    IF _eDeformStep > E_DeformationStep.nothing AND _bCamReady AND _bTeachOk THEN      // start only if previous started
      (*done during attach: 
      IF _eDeformStep < E_DeformationStep.cameraStarted THEN
        // start cam on ct
        LogLvl(Lvl:=E_LogSeverity.Debug, Msg:=F_Concat2('Start Camera with mode: ', TO_STRING(_iActiveCam.eCameraMode)));
        _pAttachedCt^.StartCamera(eCameraMode:=_iActiveCam.eCameraMode, fFeatureGrid:=_fFeatureGrid);
      *)
			IF _eDeformStep >= E_DeformationStep.cameraStarted AND _bCamStarted THEN
        // run update on ct
        // stream points
        streamPoints();
        // superview abort cases
      END_IF
      
      // NOTE: Release() is done in CamDone() method
    ELSE
      IF _bCamStarted THEN
        // error on camera while started
        LogError('Abort Camera while it was started');
			END_IF
      // release because cam not ready or pior worker not done its job
      Release(_pAttachedCt^);   // release head container
		END_IF

END_IF

// call messages
fbMsg_CamNotAvailable    (bI_Status:=bCamNotAvailable);
fbMsg_CamModeNotSupported(bI_Status:=bCamModeNotSupported);
fbMsg_CamNoConnection    (bI_Status:=NOT _bConnectionOk);
END_METHOD

END_FUNCTION_BLOCK

// ---- POUs/Print/DefGrid/FB_WorkerDefGrid.TcPOU
FUNCTION_BLOCK ABSTRACT FB_WorkerDefGrid EXTENDS FB_Worker
VAR_OUTPUT
  bError            : BOOL;                           // an error is active
  nError            : UDINT;                          // error code if error active, =0 else
END_VAR
VAR
  // config
  _pMsgConfigExt    : POINTER TO ST_MSG_CONFIG;       // external message config (puc message interface)
  _fPrintResolution : LREAL := 1;                     // print(head) resolution in [dpi]
  _fSubPxResolution : LREAL := 1;                     // SubPixel resolution [SubPx], resolution factor (fI_PrintResolution*fI_SubPxResolution=>Output resolution
  _name             : STRING;                         // Worker name
  _sVisuName        : STRING := 'VISU_WorkerDefGrid'; // Worker visu instance name
  _pEcSrc           : POINTER TO T_ErrSrc;            // Error source definition

  // job
  _bJobActive       : BOOL;                           // a job is active
  // ct
  _bAttached        : BOOL;                           // one ct is attached
  _pAttachedCt      : POINTER TO FB_ContainerDefGrid; // currently attached container (HEAD)
  _pNewAttached     : POINTER TO FB_ContainerDefGrid; // last attached container (as return value of Attach() (TAIL))
  _pNewAttachedHdlData : POINTER TO ST_WorkerDefGrid_CTData;  // pointer to handling data for last attached
  _bSupportParallelCT : BOOL := FALSE;                // support for parallel CTs (else avoid attach while one connected).
  _nAttachedCTs     : UDINT;                          // Number of currently attached CTs
  _nHeadCtId        : DINT;                           // ID of CT at Attached Head
  _pAttachedCTList  : ARRAY[nLowerIndexCTList..nUpperIndexCTList] OF POINTER TO FB_ContainerDefGrid;    // current attached CTs
  _stAttachedCTData : ARRAY[nLowerIndexCTList..nUpperIndexCTList] OF ST_WorkerDefGrid_CTData;           // additional "handling" data per attached CT
  // position control
  fCtPosition       : LREAL;     // Container position relative to worker position
  _bForceRelease    : BOOL;                           // Manually force a ct release

  // view
  nGridRowStart, nGridColStart: UDINT := 0;
END_VAR
VAR_STAT
  // static variables, SAME for ALL Workers
  _pCTM             : POINTER TO FB_CTManagerDefGrid;             // "Global" Container Manager
  _fCtSecurityReleasePos : LREAL := 0;                // [SubPx] position where to release current ct at last (security release)
END_VAR
VAR PERSISTENT
  _fWorkerPosition  : LREAL;                          // [m] worker distance to X0 (position from X0) (CT creation X0 and domain)
END_VAR
VAR CONSTANT
  // list size
  nLowerIndexCTList : UDINT := 1;
  nUpperIndexCTList : UDINT := 4; 
END_VAR

(*
  Generic abort implementation of DefGrid CT.
*)
METHOD Abort
VAR_INPUT
  iCT       : I_CT;
  sReason   : STRING;
END_VAR
VAR
  _pCt   : POINTER TO FB_ContainerDefGrid;
  eStep     : E_DeformationStep;
END_VAR
IF iCT = 0 AND _pAttachedCt <> 0 THEN             // no ct given and check if one is attached 
  _pCt := _pAttachedCt;
ELSIF getCtInst(iCT:=iCT, pCT=>_pCt) = 0 THEN     // get specific container from given interface
  RETURN; 
END_IF

IF _pCt = 0 THEN RETURN; END_IF
  
// abort CT
  // Do generic known aborts on CT
  // - Deformation
  _pCt^.getDeformationStatus(eDStep=>eStep);
  IF eStep >= E_DeformationStep.nothing THEN
    _pCt^.AbortDeformation(sReason:=sReason, Src:=_pEcSrc^, bHideLog:=FALSE);
  
END_IF
END_METHOD

METHOD PROTECTED  Attach : BOOL
VAR_INPUT
  iCT       : I_CT;            (*container at triggered event position*)
END_VAR
VAR
  i : UDINT;
END_VAR
Attach := FALSE;

IF iCT = 0 THEN
  LogError(Msg:='attach failed -> not ct given');
  
ELSIF bWorkerEnable THEN  // worker enabled
  
  IF getCtInst(iCT:=iCT, pCT=>_pNewAttached) <> 0 THEN    // get specific container
    // add to list ()
    IF push(pNewCT:=_pNewAttached) THEN 
      LogLvl(Lvl:=E_LogSeverity.Debug, Msg:=F_Concat4('Attach CT[', TO_STRING(_nAttachedCTs), ']: ', _pNewAttached^.print(0)));
      Attach:=TRUE;                                 // attach new
    END_IF
  ELSE
    LogError(Msg:='attach failed: could not get CT instance');
  END_IF

ELSIF NOT bWorkerEnable AND _nAttachedCTs > 0 THEN // disabled and already a CT attached
  // force release all attached CT, and ignore attach
  LogLvl(Lvl:=E_LogSeverity.Debug, Msg:='Worker disabled flush list of all attached CT');
  WHILE _nAttachedCTs > 0 DO
    Release(iCT:=_pAttachedCt^);
	END_WHILE

ELSIF NOT bWorkerEnable AND _pAttachedCt = 0 THEN  
  ;   // nothing to do, ignore attach

ELSE      // unspecified (error)case just log it
  LogError(Msg:='not tracked case');
END_IF


// ok to attach
END_METHOD

{attribute 'monitoring':='call'}
PROPERTY bAttached : BOOL
GET
bAttached := _bAttached;
END_GET
END_PROPERTY

{attribute 'monitoring':='call'}
PROPERTY fPosition : LREAL
GET
fPosition := _fWorkerPosition;
END_GET
SET
_fWorkerPosition := fPosition;  // [m] save position
END_SET
END_PROPERTY

(*
  Get specific container from interface.
  Returns specific container in return value and output parameter.
*)
METHOD INTERNAL getCtInst : POINTER TO FB_ContainerDefGrid
VAR_INPUT
  iCT              : I_CT;                         (*container at triggered event position*)
END_VAR
VAR_OUTPUT
  pCT              : POINTER TO FB_ContainerDefGrid;
END_VAR
IF NOT bInitialized THEN RETURN; END_IF
IF _pCTM = 0 THEN RETURN; END_IF

pCT := 0;
getCtInst := _pCTM^.GetContainerInstance(iCT);   // get real ct fb inst
IF getCtInst <> 0 THEN
  pCT := getCtInst;   // OK all good
ELSE
  LogError(Msg:='specific container not found');
END_IF
END_METHOD

(*
  Get relative position to this worker (relative to track position)
*)
METHOD getPosRelToAttach : DINT
VAR_INPUT
  iCT : I_CT;
END_VAR
// relative position to X0 - tracking offset of this worker
getPosRelToAttach := iCT.GetPosRel(iTracker:=_iCTTracker) - _nTrackOffset;
END_METHOD

METHOD Init
VAR_INPUT
  pMsgConfig : POINTER TO ST_MSG_CONFIG;         // message config
  fPrintResolution : LREAL := 1;                 // print(head) resolution in [dpi]
  fSubPxResolution : LREAL := 1;                 // SubPixel resolution [SubPx], resolution factor (fI_PrintResolution*fI_SubPxResolution=>Output resolution)
  bParallelCT : BOOL;                            // Support parallel processing of CTs
END_VAR
VAR

END_VAR
_bAttached := 0;
_pAttachedCt := 0;
_nAttachedCTs := 0;

IF _pCTM = 0 THEN LogError(Msg:='Init: invalid parameter'); RETURN; END_IF

// save config
_pMsgConfigExt := pMsgConfig;
_fPrintResolution := fPrintResolution;
_fSubPxResolution := fSubPxResolution;
_fCtSecurityReleasePos := 0;
_bSupportParallelCT := bParallelCT;

setName('');

// init error source reference
_pEcSrc := ErrorCodes.fbErrCodeMngr.registerErrSource(
  nLocId := 0,
  aInstPath := InstanceName,
  aLocDescr := _name
);
IF _pEcSrc = 0 THEN LogError('could not register error source'); END_IF

bInitialized := TRUE;
END_METHOD

METHOD ABSTRACT mJobStart
VAR_INPUT
	sJobDef	: CalmarCompPrint.I_JobDefinition;
END_VAR
// implement in parent class
END_METHOD

METHOD ABSTRACT mJobStop
VAR_INPUT
	sStatus	: CalmarCompPrint.I_JobStatus;
END_VAR
END_METHOD

PROPERTY pCTM : POINTER TO FB_CTManagerDefGrid
GET
pCTM := _pCTM;
END_GET
SET
_pCTM := pCTM;
END_SET
END_PROPERTY

METHOD PRIVATE pull : BOOL
VAR_INPUT
  pRemCT : POINTER TO FB_ContainerDefGrid;
END_VAR
VAR_OUTPUT
  nRemIndex : DINT := 0;
END_VAR
VAR
  i                : DINT;
  Index            : DINT;
  LowerIndex       : DINT := 1;
END_VAR
IF _nAttachedCTs = 0 THEN LogError('Release: but no CT is attached'); RETURN; END_IF

// -- find if ct is in attached list
Index := -1;
FOR i:= TO_DINT(nLowerIndexCTList) TO TO_DINT(nLowerIndexCTList + _nAttachedCTs - 1) DO
  IF _pAttachedCTList[i] = pRemCT THEN
    Index := i;
    EXIT;     // found
  END_IF
END_FOR
IF Index = -1 THEN LogError('Release: ct inst not found in list'); RETURN; END_IF

// do stop CT callback if removing first
IF Index = TO_DINT(nLowerIndexCTList) THEN StopCT(pCtDefGrid:=pRemCT); END_IF

// compress list
IF Index >= TO_DINT(nLowerIndexCTList) AND Index < TO_DINT(nUpperIndexCTList) THEN
  // - ct references
  MEMMOVE(              // shift all above entries down
    destAddr := ADR( _pAttachedCTList[Index] ), 
    srcAddr  := ADR( _pAttachedCTList[Index + 1] ), 
    n        := DINT_TO_UDINT(SIZEOF(_pAttachedCTList[LowerIndex]) * (UDINT_TO_DINT(_nAttachedCTs) - Index - 1 + LowerIndex))
  );
  _pAttachedCTList[nUpperIndexCTList] := 0;     // erase last(compressed) list entry
  // - ct handling data
  MEMMOVE(              // shift all above entries down
    destAddr := ADR( _stAttachedCTData[Index] ), 
    srcAddr  := ADR( _stAttachedCTData[Index + 1] ), 
    n        := DINT_TO_UDINT(SIZEOF(_stAttachedCTData[LowerIndex]) * (UDINT_TO_DINT(_nAttachedCTs) - Index - 1 + LowerIndex))
  );
  MEMSET(destAddr:=ADR(_stAttachedCTData[nUpperIndexCTList]), fillByte:=0, n:=SIZEOF(_stAttachedCTData[1]));  // erase last(compressed) list entry
END_IF
_pAttachedCTList[_nAttachedCTs] := 0;   // erase last element
MEMSET(destAddr:=ADR(_stAttachedCTData[_nAttachedCTs]), fillByte:=0, n:=SIZEOF(_stAttachedCTData[1]));  // erase last element
  
// remove
_nAttachedCTs := _nAttachedCTs - 1;   // remove one element

IF _nAttachedCTs > 0 THEN 
  // Start new HEAD
  _pAttachedCt := _pAttachedCTList[1];
  _bAttached := TRUE;
  StartCT(pCtDefGrid:=_pAttachedCt);
ELSE
  // CT list empty (no ct attached)
  _pAttachedCt := 0;
  _bAttached := 0;
END_IF

nRemIndex := Index;
pull := TRUE;
END_METHOD

METHOD PRIVATE push : BOOL
VAR_INPUT
  pNewCT : POINTER TO FB_ContainerDefGrid;
END_VAR
// checks
// - valid param
IF pNewCT = 0 THEN LogError('push: invalid pointer'); RETURN; END_IF
// - list full
IF _nAttachedCTs >= nUpperIndexCTList THEN  // list overflow no free element for processing
  LogError('Worker processing list full, ignore new CT');
  Abort(iCT:=pNewCT^, sReason:='attach failed - too many attached');  // abort new CT (no release because not yet attached)
  RETURN;
END_IF
// - only one CT allowed
IF _nAttachedCTs > 0 AND NOT _bSupportParallelCT THEN
  LogError(Msg:='another container already attached -> ignore new (set error)');
  Abort(iCT:=pNewCt^, sReason:='attach failed - no parallel support');  // abort new CT
END_IF

// add to list
_nAttachedCTs := _nAttachedCTs + 1;
_pAttachedCTList[_nAttachedCTs] := pNewCT;
MEMSET(destAddr:=ADR(_stAttachedCTData[_nAttachedCTs]), fillByte:=0, n:=SIZEOF(_stAttachedCTData[1]));  // clear additional data
_pNewAttachedHdlData := ADR(_stAttachedCTData[_nAttachedCTs]);   // select handling data for new attached ct 

// apply head
IF _nAttachedCTs = 1 THEN
  // set HEAD
  _pAttachedCt := _pAttachedCTList[nLowerIndexCTList];  
  _bAttached := TRUE;

  // start callback on HEAD
  StartCT(pCtDefGrid:=_pAttachedCt);
END_IF

push := TRUE;
END_METHOD

(*
  Release CT from Worker.
  :return: TRUE if CT was released, FALSE if no CT was registered 
*)
METHOD Release : BOOL
VAR_INPUT
  iCT              : I_CT;                         (*container at triggered event position*)
END_VAR
VAR
  nIdx             : DINT;
  pCT              : POINTER TO FB_ContainerDefGrid;
END_VAR
// remove CT -----------------------------------------------------
// -- get real instance
pCT := getCtInst(iCT:=iCT);
IF pCT = 0 THEN LogError('Release: could not find ct instance'); RETURN; END_IF

// remove and release CT
IF pull(pRemCT:=pCT, nRemIndex=>nIdx) THEN
  LogLvl(Lvl:=E_LogSeverity.Debug, Msg:=F_Concat4('Release CT[', TO_STRING(nIdx), '] ', pCt^.print(0)));
  Release := TRUE;  
END_IF
END_METHOD

(*
  Container will be released from tracker (destroyed) and not available anymore. 
*)
METHOD remove
VAR_INPUT
	(*container at triggered event position*)
	iCT	: I_CT;
END_VAR
SUPER^();

// nothing done
// We keep in internal WorkerList until work is done. CT will be removed from tracker.
END_METHOD

METHOD PRIVATE setName : BOOL
VAR_INPUT
  sName : STRING;
END_VAR
VAR
  nIdx : INT;
  bDone : BOOL;
END_VAR
IF sName = '' THEN
  // generate worker name
  _name := THIS^.InstanceName;
  WHILE NOT bDone DO
    nIdx := FIND(_name, '.');
    IF nIdx = 0 THEN bDone := TRUE; EXIT; 
    ELSE
      _name := RIGHT(_name,LEN(_name)-nIdx);
    END_IF 
  END_WHILE
ELSE
  _name := sName;  
END_IF
END_METHOD

METHOD PROTECTED StartCT
VAR_INPUT
 pCtDefGrid   : POINTER TO FB_ContainerDefGrid;
END_VAR
(* Override specific implementation in child class *)
END_METHOD

METHOD PROTECTED StopCT
VAR_INPUT
 pCtDefGrid   : POINTER TO FB_ContainerDefGrid;
END_VAR
(* Override specific implementation in child class *)
END_METHOD

METHOD  work
VAR
  i : UDINT;
  pCt : POINTER TO FB_ContainerDefGrid;
END_VAR
// set tracking offset
_nTrackOffset := F_MeterToSubPixel(fPosMeter:=fPosition, fResoSubPx:=_fPrintResolution*_fSubPxResolution);  // [pos domain] save position

//Work only with attached container
IF _nAttachedCTs = 0 THEN RETURN; END_IF

IF _pAttachedCt <> 0 AND_THEN _pAttachedCt^.pCT <> 0 THEN _nHeadCtId := _pAttachedCt^.pCT^.iId;
ELSE                                                      _nHeadCtId := 0; END_IF

FOR i:=nLowerIndexCTList TO nLowerIndexCTList + _nAttachedCTs - 1 DO
  pCt := _pAttachedCTList[i];

  // update CT position
  _stAttachedCTData[i].fPosRelToAttach := getPosRelToAttach(iCT:=pCt^);
  
  // release CT (manually)
  IF _bForceRelease THEN
    _bForceRelease := FALSE;
    pCt^.AbortDeformation(sReason:='Manually realease CT', Src:=_pEcSrc^, bHideLog:=FALSE);
    Release(iCT:=pCt^);

  // security release 
  ELSIF _fCtSecurityReleasePos > 0 AND (ABS(_stAttachedCTData[i].fPosRelToAttach) > _fCtSecurityReleasePos) THEN
    pCt^.AbortDeformation(sReason:=F_Concat2('Security released CT Id=', TO_STRING(pCt^.pCT^.iId)), Src:=_pEcSrc^, bHideLog:=FALSE);
    Release(iCT:=pCt^);
  END_IF

END_FOR
END_METHOD

END_FUNCTION_BLOCK

// ---- POUs/Print/DefGrid/FB_WorkerDefGrid_Deformation.TcPOU
FUNCTION_BLOCK FB_WorkerDefGrid_Deformation EXTENDS FB_WorkerDefGrid
VAR_INPUT
END_VAR
VAR_OUTPUT
END_VAR
VAR
  // references
  _iParamMediator : I_ParamMediator;
  
  //Worker specific configuration
  _nPrintUnitWidth            : UDINT;  // default print unit width [px]  
  _nImageWidthPx              : UDINT;  // size of the image (width)
  _nImageDepthPx              : UDINT;  // size of the image (depth)
  
  // -
  _bNewJob                    : BOOL;   // new job started 

  //Deformation status (per attached CT)
  _nDeformationProcPoints     : ARRAY[nLowerIndexCTList..nUpperIndexCTList] OF UDINT;  // available grid points on ct
  _nDeformationProcCols       : ARRAY[nLowerIndexCTList..nUpperIndexCTList] OF UDINT;  // number of already generated grid columns
  _eDeformStep                : ARRAY[nLowerIndexCTList..nUpperIndexCTList] OF E_DeformationStep;   // status deformation of ct
  _bDeformationError          : ARRAY[nLowerIndexCTList..nUpperIndexCTList] OF BOOL;   // status deformation of ct
  _bDeformationBusy           : ARRAY[nLowerIndexCTList..nUpperIndexCTList] OF BOOL;   // status deformation of ct
  _bDeformationDone           : ARRAY[nLowerIndexCTList..nUpperIndexCTList] OF BOOL;   // status deformation of ct
  _nDeformationErrorId        : ARRAY[nLowerIndexCTList..nUpperIndexCTList] OF UDINT;  // status deformation of ct
  _tDeformationExecutionTime  : ARRAY[nLowerIndexCTList..nUpperIndexCTList] OF TIME;   // status deformation of ct
  _bAborted                   : ARRAY[nLowerIndexCTList..nUpperIndexCTList] OF BOOL;   // status deformation of ct

  // ui
  eDeformTypeUi : E_DeformationType;
END_VAR 

VAR PERSISTENT
  _sDeformationGridSettings  : ST_DefGridSettings := (   // grid definition settings
                                  nGridPitchX:=GVL_Deformation.nC_DefaultGridPitch_X,   // this must match the hw config (in fpga)
                                  nGridPitchY:=GVL_Deformation.nC_DefaultGridPitch_Y,   // this must match the hw config (in fpag)
                                  eDeformationType:=E_DeformationType.NoDeformation
                             );
  _fDistToCam                : LREAL := 0.02;   // distance to cam worker 
END_VAR

METHOD PROTECTED  Attach : BOOL
VAR_INPUT
  iCT              : I_CT;                         (*container at triggered event position*)
END_VAR
VAR
  i : UDINT;
  bDeformErr : BOOL;
  eDeformStep : E_DeformationStep;
END_VAR
(*Please do enable externally in PrintModule
IF getCtInst(iCT:=iCT, pCT=>pCt) = 0 THEN    // get specific container
  RETURN;
END_IF

//-- (auto-) enable / disable worker based on mode (do before parent Attach(), is checked inside)
bWorkerEnable := _sDeformationGridSettings.eDeformationType <> E_DeformationType.NoDeformation 
                     AND SEL(pCt^.eCamMode > E_CameraMode.NoCorrection, FALSE, TRUE);
*)

// -- Attach
IF NOT SUPER^.Attach(iCT:=iCT) THEN
  RETURN;
END_IF

// Additional worker checks
IF _pNewAttached = 0 THEN RETURN; END_IF

// - Additional worker checks
bDeformErr := _pNewAttached^.getDeformationStatus(eDStep=>eDeformStep);   // get latest status 
  
// - deformation started? and no deformation error so far
IF bDeformErr OR eDeformStep < E_DeformationStep.cameraStarted THEN
  Release(iCT:=iCT);  // nothing to do anymore

  // - job is valid?
ELSIF _pNewAttached^.pJob = 0 OR NOT _bJobActive THEN
  _pNewAttached^.AbortDeformation(sReason:='No valid job', Src:=_pEcSrc^, bHideLog:=FALSE);
  Release(iCT:=iCT);
  
// - did camera start?  
(*ELSIF eDeformStep < E_DeformationStep.cameraStarted THEN
  _pNewAttached^.AbortDeformation(sReason:='Prio steps did not start', Src:=_pEcSrc^);
  Release(iCT:=iCT);
*)
  
// - OK attach
ELSE
  // checks
  IF eDeformStep < E_DeformationStep.cameraStarted THEN LogWarning('Sub-optimal timing, camera did not yet start'); END_IF
  // start deformation
  _pNewAttached^.StartDeformation(
    sDefGridSettings:=_sDeformationGridSettings, 
    fStartDeformationPos:=getPosRelToAttach(iCT)/_fSubPxResolution   // [px]
  );
  Attach := TRUE;
END_IF
END_METHOD

METHOD InitWorkerDeformation : BOOL
VAR_INPUT
  nPrintUnitWidth : UDINT;
  iDefGridParamMediator : I_ParamMediator;
END_VAR
VAR
  i : UDINT;
END_VAR
IF NOT bInitialized THEN LogError('Base Worker not initialized! call init() before'); RETURN; END_IF
IF iDefGridParamMediator = 0 THEN bInitialized := FALSE; LogError('Invalid parameter, no valid param mediator'); RETURN; END_IF


// worker specific init
_nPrintUnitWidth := nPrintUnitWidth;
_iParamMediator := iDefGridParamMediator;
_bNewJob := FALSE;

FOR i:=nLowerIndexCTList TO nUpperIndexCTList DO
  _nDeformationProcPoints[i]     := 0;
  _nDeformationProcCols[i]       := 0;
  _eDeformStep[i]                := 0;
  _bDeformationError[i]          := 0;
  _bDeformationBusy[i]           := 0;
  _bDeformationDone[i]           := 0;
  _nDeformationErrorId[i]        := 0;
  _tDeformationExecutionTime[i]  := T#0S;
  _bAborted[i]                   := 0;
END_FOR
END_METHOD

METHOD mJobStart
VAR_INPUT
	sJobDef	: CalmarCompPrint.I_JobDefinition;
END_VAR
VAR
  sCamSettings : ST_CameraGridSettings;
END_VAR
// check and init invalid settings
IF _iParamMediator = 0 THEN LogError('no parameter mediator'); RETURN; END_IF
IF _sDeformationGridSettings.nGridPitchX = 0 THEN _sDeformationGridSettings.nGridPitchX:=GVL_Deformation.nC_DefaultGridPitch_X; LogError(F_Concat2('nGridPitchX not configured, set default=', TO_STRING(GVL_Deformation.nC_DefaultGridPitch_X))); END_IF
IF _sDeformationGridSettings.nGridPitchY = 0 THEN _sDeformationGridSettings.nGridPitchY:=GVL_Deformation.nC_DefaultGridPitch_Y; LogError(F_Concat2('nGridPitchY not configured, set default=', TO_STRING(GVL_Deformation.nC_DefaultGridPitch_Y))); END_IF
IF _nPrintUnitWidth = 0 THEN LogError('_nPrintUnitWidth not configured'); END_IF
IF fPosition = 0 THEN LogError('No valid Worker position: set it to WorkerCamera.fCameraToPrintOffset + 0.05; '); END_IF

// configuration
// calculate deformation  settings
// - save image y-offset (centered)
// - save image size
_nImageWidthPx := DINT_TO_UDINT(F_MeterToSubPixel(fPosMeter:=sJobDef.fImageWidth/1000, fResoSubPx:=_fPrintResolution));
_nImageDepthPx := DINT_TO_UDINT(F_MeterToSubPixel(fPosMeter:=sJobDef.fImageDepth/1000, fResoSubPx:=_fPrintResolution));
_sDeformationGridSettings.nGridImageOffsetY := LIMIT(0, ((_nPrintUnitWidth - _nImageWidthPx)) / 2, (_nPrintUnitWidth));  // TODO: if you can get this value from PUC use the other one to have a consistent image shift value 

// - calc grid size and number of points
(*
  Use image width / depth in px divide by GridPitch in X/Y to do a ceil(always next bigger integer).
  +1 -> Because Grid starts at 0 until the calculated numbers we have one point more [0, 1, 2, 3] = 4 points (not 3) 
*)
IF _sDeformationGridSettings.nGridPitchX > 0 AND _sDeformationGridSettings.nGridPitchY > 0 THEN
  _sDeformationGridSettings.nGridSizeX := F_Ceil(val:=UDINT_TO_LREAL(_nImageDepthPx)/_sDeformationGridSettings.nGridPitchX) + 1;
  _sDeformationGridSettings.nGridSizeY := F_Ceil(val:=UDINT_TO_LREAL(_nImageWidthPx + _sDeformationGridSettings.nGridImageOffsetY)/_sDeformationGridSettings.nGridPitchY) + 1;
END_IF
_sDeformationGridSettings.nGridPoints :=  _sDeformationGridSettings.nGridSizeX * _sDeformationGridSettings.nGridSizeY;

sCamSettings := _iParamMediator.sCameraGridSettings;
_sDeformationGridSettings.eDeformationType := sCamSettings.eDeformationType;   // apply deformation mode (for ui)
eDeformTypeUi := _sDeformationGridSettings.eDeformationType;

_bJobActive := TRUE;
END_METHOD

METHOD  mJobStop
VAR_INPUT
	sStatus	: CalmarCompPrint.I_JobStatus;
END_VAR
_bJobActive := FALSE;
END_METHOD

(*
  Release CT from Worker.
  :return: TRUE if CT was released, FALSE if no CT was registered 
*)
METHOD Release : BOOL
VAR_INPUT
  iCT              : I_CT;                         (*container at triggered event position*)
END_VAR
VAR
  i                : DINT;
  Index            : DINT;
  LowerIndex       : DINT := 1;
  pCt              : POINTER TO FB_ContainerDefGrid;
  eStep            : E_DeformationStep;
END_VAR
IF iCT = 0 OR _nAttachedCTs = 0 THEN RETURN; END_IF

// release from deformation module
IF getCtInst(iCT:=iCT, pCT=>pCt) = 0 THEN LogError('Release: could not find ct instance'); RETURN; END_IF
IF _iParamMediator <> 0 THEN
  pCt^.getDeformationStatus(eDStep => estep);
  IF estep >= E_DeformationStep.createdScriptContainer THEN
    pCt^.StopScript(iCT:=iCT);
    //_pParamMediator^.ReleaseDeformationCT(iCT:=iCT);
  END_IF
END_IF

Release := SUPER^.Release(iCT:=iCT);
END_METHOD

PROPERTY sDeformationGridSettings : ST_DefGridSettings
GET
sDeformationGridSettings := _sDeformationGridSettings;
END_GET
END_PROPERTY

METHOD setupPosition
VAR
  sCamSettings : ST_CameraGridSettings;
END_VAR
IF _pAttachedCt <> 0 THEN RETURN; END_IF    // Update only without attached container

sCamSettings := _iParamMediator.sCameraGridSettings;

// set tracking offset
fPosition := sCamSettings.fDetectToCam + _fDistToCam;
END_METHOD

METHOD  work
VAR
  i : UDINT;
  pCT : POINTER TO FB_ContainerDefGrid;
END_VAR
//-----------------------------------------------------------
SUPER^.work();      // Parent implementation

setupPosition();    // Worker position update

// Work only with attached container (additional work to Base class)
FOR i:=nLowerIndexCTList TO nLowerIndexCTList + _nAttachedCTs - 1 DO
  pCt := _pAttachedCTList[i];
 
  // update deformation handler
  pCT^.UpdateDeformation(fPos:=_stAttachedCTData[i].fPosRelToAttach/_fSubPxResolution);  // pos in [px]
  
  // get status
  _bDeformationError[i] := pCt^.getDeformationStatus(eDStep => _eDeformStep[i], 
                            bBusy => _bDeformationBusy[i],
                            bDone => _bDeformationDone[i],
                            nErrorId => _nDeformationErrorId[i], 
                            tExecutionTime => _tDeformationExecutionTime[i],
                            bAborted => _bAborted[i]);
  _nDeformationProcPoints[i] := pCt^.nAvailableGridPoints;
  _nDeformationProcCols[i]   := pCt^.nAvailableGridCols;
     
  // Release container when all points have been processed or error
  IF _bDeformationDone[i] OR _bDeformationError[i] THEN
    // tag CT with error if deformation had an error
    IF _bDeformationError[i] THEN 
      IF NOT _bAborted[i] THEN
        pCt^.AbortDeformation(sReason:=F_Concat2('WorkerDeformation: ', EC_DefGrid.ecDefGrid_DefGridError.Desc), Src:=_pEcSrc^, bHideLog:=FALSE);
      //not needed ELSE
      //  pCt^.setError(ErrDef:=EC_DefGrid.ecDefGrid_DefGridError, Src:=_pEcSrc^);
      END_IF
    END_IF
    LogLvl(Lvl:=E_LogSeverity.Detail, Msg:=F_Concat4('Done with: CamP=',  TO_STRING(pCT^.nRegisteredCameraPoints), ' GridP=', TO_STRING(pCt^.nAvailableGridPoints)));
    Release(pCt^);
  END_IF
  
END_FOR
END_METHOD

END_FUNCTION_BLOCK

// ---- POUs/Print/DefGrid/FB_DropSpeedComp.TcPOU
FUNCTION_BLOCK FB_DropSpeedComp
VAR_INPUT
  fMasterSpeed         : LREAL; //[m/s]
  fDropTravelDistance  : LREAL; //[m]
END_VAR
VAR_OUTPUT
  fDropPlacementError  : LREAL;
END_VAR
VAR PERSISTENT
  _bEnable             : BOOL := TRUE;
  _fDropSpeed          : LREAL := 6;         //[m/s] DropSpeed compensation, drop speed
  _fDropSpeedDeadTime  : LREAL := 0.388889;  //[ms]  DropSpeed compensation, additional dead time
END_VAR
VAR
  bCalcDeadTime        : BOOL;
  fTestSpeed           : ARRAY[1..2] OF LREAL;  // [m/min] speed at which test was done [SpeedTest1, SpeedTest2]
  fTestDisplacement    : ARRAY[1..2] OF LREAL;  // [um] measured displacement after test [MesureTest1, MeasureTest2]
  fDiffSpeed : LREAL;
  fDiffPlace : LREAL;
END_VAR

(*Speed compensation*)
IF _bEnable AND (_fDropSpeed > 0) THEN
	fDropPlacementError :=  (  (fDropTravelDistance / _fDropSpeed)
                        + (_fDropSpeedDeadTime / 1000))             (*[s]*)
                        * fMasterSpeed;
ELSE
  fDropPlacementError := 0;
END_IF;

// calculate add/dead time
IF bCalcDeadTime THEN bCalcDeadTime := FALSE;
  calcDeadTime();
END_IF

{attribute 'monitoring':='call'}
PROPERTY bEnable : BOOL
GET
bEnable := _bEnable;
END_GET
SET
_bEnable := bEnable;
END_SET
END_PROPERTY

METHOD PRIVATE calcDeadTime : BOOL
VAR_INPUT
END_VAR
fDiffSpeed :=  ( fTestSpeed[2] - fTestSpeed[1] ) * 1/60;
fDiffPlace :=  ( fTestDisplacement[2] - fTestDisplacement[1] ) * 1/1_000_000;

IF fDiffSpeed <> 0 THEN   // avoid crash
  // calc time
  _fDropSpeedDeadTime := 
  (
      fDiffPlace      // displacement diff
    * 1/fDiffSpeed    // speed diff
  ) * 1000;           // [s] -> [ms]
ELSE
  F_LogError('DropSpeedComp invalid TestSpeed given -> DeadTime not updated');
END_IF


// reset entries
fTestSpeed[2] := fTestSpeed[1] := 0;
fTestDisplacement[2] := fTestDisplacement[1] := 0;
END_METHOD

{attribute 'monitoring':='call'}
PROPERTY fDropSpeed : LREAL
GET
fDropSpeed := _fDropSpeed;
END_GET
SET
_fDropSpeed := fDropSpeed;
END_SET
END_PROPERTY

{attribute 'monitoring':='call'}
PROPERTY fDropSpeedDeadTime : LREAL
GET
fDropSpeedDeadTime := _fDropSpeedDeadTime;
END_GET
SET
_fDropSpeedDeadTime := fDropSpeedDeadTime;
END_SET
END_PROPERTY

END_FUNCTION_BLOCK

// ---- POUs/Print/DefGrid/FB_FineAlignement.TcPOU
(*
  This fb handles mechanical print unit corrections.
  - a 4p grid distortion
  - print unit bar banana correction
  NOTE: temperature extention of whole printbar is still handled in camera
*)
FUNCTION_BLOCK FB_FineAlignement EXTENDS FB_BasePrint IMPLEMENTS I_GridPointCorrection
VAR
  // config
  _fPxResolution     : LREAL; // pixel resolution

  // corrections
  //-- 4 point PU deformation correction/distortion
  //    VISU setup point providing reference and correction (NOTE: persists settings internally)
  _fbPlcCorrPoints : ARRAY[1..4] OF FB_PointCorr;
  //-- banana correction
  _fT1 : LREAL;   // temperature 1
  _fT2 : LREAL;   // temperature 2
  _dx_middle : LREAL;  // correction in middle (for view only)
  _y_max : LREAL; // print unit width [mm]
  //-- PUC 4p correction
  _pAdsCam           : POINTER TO FB_ADS_CAMERA;  // camera interface PUC
  aPucPointNames : ARRAY[1..4] OF STRING := ['1','2','3','4'];
  
  // helper
  lCtr     : UDINT;
  
  // unit test & debug
  _bUT_4p, _bUT_banana, _bUT_4pPuc : BOOL;
  _sUTPoints_dx : ARRAY[0..nC_UT_cols, 0..nC_UT_rows] OF LREAL;
  _sUTPoints_dy : ARRAY[0..nC_UT_cols, 0..nC_UT_rows] OF LREAL;
  // 4pPUC
  bSelect : ARRAY[1..4] OF BOOL;
  bSelected : ARRAY[1..4] OF BOOL;
  nSelectedPoint : UDINT;
  bXPlus, bXMinus, bYPlus, bYMinus : BOOL;
END_VAR
VAR PERSISTENT
  //-- 4point correction
  _bEnable_4p    : BOOL := FALSE;
  _bEnablePuc_4p : BOOL := FALSE;
  //  persistence of points see: FB_PointCorr
  //-- banana correction
  _bEnable_banana : BOOL := FALSE;
  _e_max_per_deltaT : LREAL := 0.01;  // [mm/°C]  TODO: use from config
END_VAR
VAR CONSTANT
  // Unit test configuration
  nC_UT_cols : DINT := 6;   // for test only
  nC_UT_rows : DINT := 5;   // for test only
END_VAR

// cyclic caluclation and view updates
//        NOTE: deformation is happening in updateCorrection() callback

//-- 4p correction
//   visu overrides (limitation rectancular point definition)
_fbPlcCorrPoints[3].fX_Ref := _fbPlcCorrPoints[1].fX_Ref;
_fbPlcCorrPoints[4].fX_Ref := _fbPlcCorrPoints[2].fX_Ref;
_fbPlcCorrPoints[2].fY_Ref := _fbPlcCorrPoints[1].fY_Ref;
_fbPlcCorrPoints[4].fY_Ref := _fbPlcCorrPoints[3].fY_Ref;
//   update CorrectionPoints view elements
FOR lCtr := 1 TO 4 DO
  _fbPlcCorrPoints[lCtr](); 
END_FOR

//-- banana correction
// just calculate the dx in the middle of the PU, just for the VISU
calc_banana_correction(x_pos:=0, y_pos:=_y_max/(2*1000), fT1:=_fT1, fT2:=_fT2, dx_corr=>_dx_middle);
_dx_middle := _dx_middle * 1000; // [m] --> [mm] for visu

// Unit test
IF _bUT_4p THEN _bUT_4p := FALSE; _test_4p(); END_IF
IF _bUT_banana THEN _bUT_banana := FALSE; _test_banana(); END_IF
IF _bUT_4pPuc THEN _test_Puc4p(); END_IF

METHOD PRIVATE _test_4p
VAR
  sPoint : ST_DeformationPoint;
  nCol, nRow, nCrPoint : DINT;
  dx, dy : LREAL;       // correction in [m]
  dx_px, dy_px : DINT;  // correction in [px]
  pPUC_CorrPointsInd : POINTER TO ARRAY[1..4] OF ST_CORRECTION_POINT;
  
  nCorrectionX : ARRAY[1..4] OF REAL := [-0.25, -0.2, 0.35, 0.35];
  nCorrectionY : ARRAY[1..4] OF REAL := [-0.45, -0.3, -0.8, -0.65];
  nCorrectionPointX_PLC : ARRAY[1..4] OF REAL := [0, 1000,   0, 1000];
  nCorrectionPointY_PLC : ARRAY[1..4] OF REAL := [0,   0, 702, 702];
  nCorrectionPointX_PUC : ARRAY[1..4] OF REAL := [0, 671.99,   0, 671.99];
  nCorrectionPointY_PUC : ARRAY[1..4] OF REAL := [-0.0001666666, -0.0001666666, 754.2108, 754.2108];
END_VAR
// setup test correcton points location for PLC & PUC 4p testing
pPUC_CorrPointsInd := _pAdsCam^.pCorrectionPointsIndication;
IF pPUC_CorrPointsInd = 0 THEN F_Report_Error(ErrType:=EN_REPORT_ERROR_TYPE.Report_Error_0Pointer);  RETURN; END_IF

FOR nCrPoint:=1 TO 4 DO
  // correction point location
  // -- PLC
  _fbPlcCorrPoints[nCrPoint].fX_Ref := nCorrectionPointX_PLC[nCrPoint];
  _fbPlcCorrPoints[nCrPoint].fY_Ref := nCorrectionPointY_PLC[nCrPoint];
  // -- PUC  
  pPUC_CorrPointsInd^[nCrPoint].posx := nCorrectionPointX_PUC[nCrPoint];
  pPUC_CorrPointsInd^[nCrPoint].posy := nCorrectionPointY_PUC[nCrPoint];
  
  // point correction  
  // -- PLC
  _fbPlcCorrPoints[nCrPoint].fX := nCorrectionX[nCrPoint];
  _fbPlcCorrPoints[nCrPoint].fY := nCorrectionY[nCrPoint];
  // -- PUC
  pPUC_CorrPointsInd^[nCrPoint].x := nCorrectionX[nCrPoint];
  pPUC_CorrPointsInd^[nCrPoint].y := nCorrectionY[nCrPoint];
END_FOR

// generate internal test grid
FOR nCol:=0 TO nC_UT_cols DO
  FOR nRow:=0 TO nC_UT_rows DO
    sPoint.col := nCol;
    sPoint.row := nRow;
    sPoint.x_ref := nCol * TO_DINT(GVL_Deformation.nC_DefaultGridPitch_X);
    sPoint.y_ref := nRow * TO_DINT(GVL_Deformation.nC_DefaultGridPitch_Y);
    sPoint.dx := 0;   // no previous deformation
    sPoint.dy := 0;   // no previous deformation
    
    // calc 4p PLC correction and apply to point
    calc_4p_correction(
        x_pos:=F_SubPixelToMeter(lPosSubPx:=sPoint.x_ref, fResSubPx:=_fPxResolution), 
        y_pos:=F_SubPixelToMeter(lPosSubPx:=sPoint.y_ref, fResSubPx:=_fPxResolution), 
        dx_corr=>dx, 
        dy_corr=>dy);
    LogInfo(
      F_Concat4(
        '4p PLC: point:', 
        F_Concat4(' x=', TO_STRING(sPoint.x_ref), '/y=', TO_STRING(sPoint.y_ref)),
        F_Concat2(' dx=', TO_STRING(dx)),
        F_Concat2(' dy=', TO_STRING(dy))
      )
    );

    // --- store in table for verification with Excel caluculation
    dx_px := F_MeterToSubPixel(fPosMeter:=dx, fResoSubPx:=_fPxResolution);
    dy_px := F_MeterToSubPixel(fPosMeter:=dy, fResoSubPx:=_fPxResolution);
    // save corrected point
    _sUTPoints_dx[nCol, nRow] := dx_px;
    _sUTPoints_dy[nCol, nRow] := dy_px;
    // print corrected point
    LogInfo(
      F_Concat4(
        F_Concat4('[c/r] ', TO_STRING(sPoint.col), '/', TO_STRING(sPoint.row)),
        F_Concat7(' dx: ', TO_STRING(sPoint.dx), '>', TO_STRING(dx_px), ' (', TO_STRING(dx), ')'),
        F_Concat7(' dy: ', TO_STRING(sPoint.dy), '>', TO_STRING(dy_px), ' (', TO_STRING(dy), ')'),
        SEL(sPoint.dx<>dx_px OR sPoint.dy<>dy_px,'',' !!!')
      )
    );
    // ---------------------------------
    
    // calc 4p PUC correction and apply to point
    calc_PUC_4p_correction(
        x_pos:=F_SubPixelToMeter(lPosSubPx:=sPoint.x_ref, fResSubPx:=_fPxResolution), 
        y_pos:=F_SubPixelToMeter(lPosSubPx:=sPoint.y_ref, fResSubPx:=_fPxResolution), 
        dx_corr=>dx, 
        dy_corr=>dy);
    LogInfo(
      F_Concat4(
        '4p PUC: point:', 
        F_Concat4(' x=', TO_STRING(sPoint.x_ref), '/y=', TO_STRING(sPoint.y_ref)),
        F_Concat2(' dx=', TO_STRING(dx)),
        F_Concat2(' dy=', TO_STRING(dy))
      )
    );

  END_FOR  
END_FOR
END_METHOD

METHOD PRIVATE _test_banana
VAR
  sPoint : ST_DeformationPoint;
  nCol, nRow : DINT;
  dx, dy : LREAL;       // correction in [m]
  dx_px, dy_px : LREAL;  // correction in [px]
END_VAR
// generate internal grid
FOR nCol:=0 TO nC_UT_cols DO
  FOR nRow:=0 TO nC_UT_rows DO
    sPoint.col := nCol;
    sPoint.row := nRow;
    sPoint.x_ref := nCol * TO_DINT(GVL_Deformation.nC_DefaultGridPitch_X);
    sPoint.y_ref := nRow * TO_DINT(GVL_Deformation.nC_DefaultGridPitch_Y);
    sPoint.dx := 0;   // no previous deformation
    sPoint.dy := 0;   // no previous deformation
    
    // calc correction and apply to point
    calc_banana_correction(
        x_pos:=F_SubPixelToMeter(lPosSubPx:=sPoint.x_ref, fResSubPx:=_fPxResolution), 
        Y_pos:=F_SubPixelToMeter(lPosSubPx:=sPoint.y_ref, fResSubPx:=_fPxResolution),
        fT1 := 68,
        fT2 := 48, 
        dx_corr=>dx
    );
    dx_px := dx;
    dy_px := dy;
    // save corrected point (dx @y-pos)
    _sUTPoints_dx[nCol, nRow] := dx_px;
    _sUTPoints_dy[nCol, nRow] := F_SubPixelToMeter(lPosSubPx:=sPoint.y_ref, fResSubPx:=_fPxResolution)*1000;
    
    // print corrected point
    LogInfo(
      F_Concat4(
        F_Concat4('[c/r] ', TO_STRING(sPoint.col), '/', TO_STRING(sPoint.row)),
        F_Concat6(' dx: ', TO_STRING(sPoint.dx), '>', TO_STRING(TO_DINT(dx_px)), ' [', TO_STRING(dx)),
        F_Concat6('  dy: ', TO_STRING(sPoint.dy), '>', TO_STRING(TO_DINT(dy_px)), ' [', TO_STRING(dy)),
        SEL(sPoint.dx<>dx_px OR sPoint.dy<>dy_px,'',' !!!')
      )
    );
  END_FOR  
END_FOR
END_METHOD

METHOD PRIVATE _test_Puc4p
VAR
  i : UDINT;

  pPUC_CorrPointsInd : POINTER TO ARRAY[1..4] OF ST_CORRECTION_POINT;
  pPoint : POINTER TO ST_CORRECTION_POINT;
END_VAR
pPUC_CorrPointsInd := _pAdsCam^.pCorrectionPointsIndication;      // get points array from ADS
IF pPUC_CorrPointsInd = 0 THEN F_Report_Error(ErrType:=EN_REPORT_ERROR_TYPE.Report_Error_0Pointer);  RETURN; END_IF

// do selection
IF    bSelect[1] THEN bSelect[1]:=FALSE; MEMSET(destAddr:=ADR(bSelected), fillByte:=0, n:=SIZEOF(bSelected)); bSelected[1] := TRUE; nSelectedPoint:=1;
ELSIF bSelect[2] THEN bSelect[2]:=FALSE; MEMSET(destAddr:=ADR(bSelected), fillByte:=0, n:=SIZEOF(bSelected)); bSelected[2] := TRUE; nSelectedPoint:=2;
ELSIF bSelect[3] THEN bSelect[3]:=FALSE; MEMSET(destAddr:=ADR(bSelected), fillByte:=0, n:=SIZEOF(bSelected)); bSelected[3] := TRUE; nSelectedPoint:=3;
ELSIF bSelect[4] THEN bSelect[4]:=FALSE; MEMSET(destAddr:=ADR(bSelected), fillByte:=0, n:=SIZEOF(bSelected)); bSelected[4] := TRUE; nSelectedPoint:=4;
END_IF

IF    bSelected[1] THEN pPoint := ADR(pPUC_CorrPointsInd^[1]);
ELSIF bSelected[2] THEN pPoint := ADR(pPUC_CorrPointsInd^[2]);
ELSIF bSelected[3] THEN pPoint := ADR(pPUC_CorrPointsInd^[3]);
ELSIF bSelected[4] THEN pPoint := ADR(pPUC_CorrPointsInd^[4]);
ELSE                    pPoint := ADR(pPUC_CorrPointsInd^[1]);
END_IF

IF bXPlus  THEN bXPlus  := FALSE; pPoint^.x := pPoint^.x + 0.05; END_IF
IF bXMinus THEN bXMinus := FALSE; pPoint^.x := pPoint^.x - 0.05; END_IF
IF bYPlus  THEN bYPlus  := FALSE; pPoint^.y := pPoint^.y + 0.05; END_IF
IF bYMinus THEN bYMinus := FALSE; pPoint^.y := pPoint^.y - 0.05; END_IF
END_METHOD

(*
  Calculate grid point displacement for a distortion with 4 rectangular defined points.
  Uses 2-bilinear interpolation between the 4 rectancular reference points.
*)
METHOD PRIVATE calc_4p_correction : BOOL
VAR_INPUT
  x_pos   : LREAL;    // point x position [m]
  y_pos   : LREAL;    // point y position [m]
END_VAR
VAR_OUTPUT
  dx_corr : LREAL;    // point correction x [m]
  dy_corr : LREAL;    // point correction y [m]
END_VAR
VAR
  dx, dy : LREAL;     // difference between Calibration Points (rectangle)
  x1, x2, y1, y2 : LREAL;
  cx1, cx2, cy1, cy2 : LREAL;
  GPx, GPy : LREAL;
  CVx, CVy : LREAL;
  lErrCtr : UDINT;
END_VAR

// Grid point position
GPx := x_pos; 
GPy := y_pos;

// Interpolation in x
x1 := _fbPlcCorrPoints[1].fX_Ref / 1000;    // [mm -> m]
x2 := _fbPlcCorrPoints[2].fX_Ref / 1000;    // [mm -> m]
dx := x2-x1;
IF dx = 0 THEN (*F_Report_Error(ErrType:=EN_REPORT_ERROR_TYPE.Report_Error_0Pointer);*) RETURN; END_IF

cx1 := (x2-GPx)/dx * (_fbPlcCorrPoints[1].fX / 1000) + (GPx-x1)/dx * (_fbPlcCorrPoints[2].fX / 1000);
cx2 := (x2-GPx)/dx * (_fbPlcCorrPoints[3].fX / 1000) + (GPx-x1)/dx * (_fbPlcCorrPoints[4].fX / 1000);
cy1 := (x2-GPx)/dx * (_fbPlcCorrPoints[1].fY / 1000) + (GPx-x1)/dx * (_fbPlcCorrPoints[2].fY / 1000);
cy2 := (x2-GPx)/dx * (_fbPlcCorrPoints[3].fY / 1000) + (GPx-x1)/dx * (_fbPlcCorrPoints[4].fY / 1000);

// Interpolation in y
y1 := _fbPlcCorrPoints[1].fY_Ref / 1000;    // [mm -> m]
y2 := _fbPlcCorrPoints[3].fY_Ref / 1000;    // [mm -> m]
dy := y2-y1;
IF dy = 0 THEN (*F_Report_Error(ErrType:=EN_REPORT_ERROR_TYPE.Report_Error_0Pointer);*) RETURN; END_IF

// Calc interpolated 
CVx := (y2 - GPy)/dy * cx1 + (GPy-y1)/dy * cx2;
CVy := (y2 - GPy)/dy * cy1 + (GPy-y1)/dy * cy2;

// return accurate new correction only
dx_corr := CVx;
dy_corr := CVy;

calc_4p_correction := TRUE;
END_METHOD

(*
  Calculate grid point displacement for print unit banana deformation.
  2nd order approximation.
*)
METHOD PRIVATE calc_banana_correction : BOOL
VAR_INPUT
  x_pos   : LREAL;    // point x position [m]
  y_pos   : LREAL;    // point y position [m]
  fT1     : LREAL;    // temperature 1 [°C]
  fT2     : LREAL;    // temperature 2 [°C]
END_VAR
VAR_OUTPUT
  dx_corr : LREAL;    // point correction x [m]
END_VAR
VAR
  delta_T : LREAL;   // delta temperature
  e_max   : LREAL;   //
  a : LREAL;
  x_dash, y_dash : LREAL;
END_VAR
IF _y_max = 0 THEN RETURN; END_IF

x_dash := y_pos * 1000; // [m] -> [mm]

delta_T := fT2-fT1;
e_max   := delta_T * _e_max_per_deltaT;

a := 4 * e_max /  EXPT(_y_max, 2);
y_dash := a * EXPT(x_dash - (_y_max / 2), 2) - e_max;

// correction value
dx_corr := (y_dash / 1000);  // [mm] -> [m]

calc_banana_correction := TRUE;
END_METHOD

(*
  Calculate grid point displacement for a distortion with 4 rectangular defined points.
  Uses 2-bilinear interpolation between the 4 rectancular reference points.
*)
METHOD PRIVATE calc_PUC_4p_correction : BOOL
VAR_INPUT
  x_pos   : LREAL;    // point x position [m]
  y_pos   : LREAL;    // point y position [m]
END_VAR
VAR_OUTPUT
  dx_corr : LREAL;    // point correction x [m]
  dy_corr : LREAL;    // point correction y [m]
END_VAR
VAR
  dx, dy : LREAL;     // difference between Calibration Points (rectangle)
  x1, x2, y1, y2 : LREAL;
  cx1, cx2, cy1, cy2 : LREAL;
  GPx, GPy : LREAL;
  CVx, CVy : LREAL;
  lErrCtr : UDINT;
  
  pPUC_CorrPointsInd : POINTER TO ARRAY[1..4] OF ST_CORRECTION_POINT;
END_VAR
VAR CONSTANT
  fTranslateX : REAL := 1;
  fTranslateY : REAL := -1;
END_VAR
pPUC_CorrPointsInd := _pAdsCam^.pCorrectionPointsIndication;      // get points array from ADS
IF pPUC_CorrPointsInd = 0 THEN F_Report_Error(ErrType:=EN_REPORT_ERROR_TYPE.Report_Error_0Pointer);  RETURN; END_IF

// NOTE: the anchor points (poyx,posy) of the PUC points are set in WorkerCamera.mJobStart!

// Grid point position
GPx := x_pos; 
GPy := y_pos;

// Interpolation in x
x1 := pPUC_CorrPointsInd^[1].posx / 1000;    // [mm -> m]
x2 := pPUC_CorrPointsInd^[2].posx / 1000;    // [mm -> m]
dx := x2-x1;
IF dx = 0 THEN (*F_Report_Error(ErrType:=EN_REPORT_ERROR_TYPE.Report_Error_0Pointer);*) RETURN; END_IF

cx1 := (x2-GPx)/dx * ((pPUC_CorrPointsInd^[1].x * fTranslateX) / 1000) + (GPx-x1)/dx * ((pPUC_CorrPointsInd^[2].x * fTranslateX) / 1000);
cx2 := (x2-GPx)/dx * ((pPUC_CorrPointsInd^[3].x * fTranslateX) / 1000) + (GPx-x1)/dx * ((pPUC_CorrPointsInd^[4].x * fTranslateX) / 1000);
cy1 := (x2-GPx)/dx * ((pPUC_CorrPointsInd^[1].y * fTranslateY) / 1000) + (GPx-x1)/dx * ((pPUC_CorrPointsInd^[2].y * fTranslateY) / 1000);
cy2 := (x2-GPx)/dx * ((pPUC_CorrPointsInd^[3].y * fTranslateY) / 1000) + (GPx-x1)/dx * ((pPUC_CorrPointsInd^[4].y * fTranslateY) / 1000);

// Interpolation in y
y1 := pPUC_CorrPointsInd^[1].posy / 1000;    // [mm -> m]
y2 := pPUC_CorrPointsInd^[3].posy / 1000;    // [mm -> m]
dy := y2-y1;
IF dy = 0 THEN (*F_Report_Error(ErrType:=EN_REPORT_ERROR_TYPE.Report_Error_0Pointer);*) RETURN; END_IF

// Calc interpolated 
CVx := (y2 - GPy)/dy * cx1 + (GPy-y1)/dy * cx2;
CVy := (y2 - GPy)/dy * cy1 + (GPy-y1)/dy * cy2;

// return accurate new correction only
dx_corr := CVx;
dy_corr := CVy;

calc_PUC_4p_correction := TRUE;
END_METHOD

PROPERTY fT_PL1 : LREAL
SET
_fT1 := fT_PL1;
END_SET
END_PROPERTY

PROPERTY fT_PL2 : LREAL
SET
_fT2 := fT_PL2;
END_SET
END_PROPERTY

METHOD init : BOOL
VAR_INPUT
  pAdsCam        : POINTER TO FB_ADS_CAMERA;  // camera interface PUC
  fPxReso        : LREAL;   // pixel resolution
  fPuWidth       : LREAL;   // Print unit width [m]
END_VAR
_fPxResolution := fPxReso;
_y_max         := fPuWidth * 1000;  // -> [mm]
_pAdsCam       := pAdsCam;
IF _pAdsCam = 0 THEN LogError('missing _pAdsCam, ads interface unknown, call worker specific init before'); END_IF

// PU Deformation
_fbPlcCorrPoints[1].init(aName:='P1', aUnit:='mm', fX_Min:=-5, fX_Max:=5, fY_Min:=-5, fY_Max:=5, fIncrStep:=0.05, 
                        bButnInvertX:=TRUE, bButnInvertY:=TRUE, bValInvertX:=TRUE, bValInvertY:=FALSE);
_fbPlcCorrPoints[2].init(aName:='P2', aUnit:='mm', fX_Min:=-5, fX_Max:=5, fY_Min:=-5, fY_Max:=5, fIncrStep:=0.05,
                        bButnInvertX:=TRUE, bButnInvertY:=TRUE, bValInvertX:=TRUE, bValInvertY:=FALSE);
_fbPlcCorrPoints[3].init(aName:='P3', aUnit:='mm', fX_Min:=-5, fX_Max:=5, fY_Min:=-5, fY_Max:=5, fIncrStep:=0.05,
                        bButnInvertX:=TRUE, bButnInvertY:=TRUE, bValInvertX:=TRUE, bValInvertY:=FALSE);
_fbPlcCorrPoints[4].init(aName:='P4', aUnit:='mm', fX_Min:=-5, fX_Max:=5, fY_Min:=-5, fY_Max:=5, fIncrStep:=0.05,
                        bButnInvertX:=TRUE, bButnInvertY:=TRUE, bValInvertX:=TRUE, bValInvertY:=FALSE);
END_METHOD

(*
  Apply fine-alignement corrections to DefGrid point
*)
METHOD updateCorrection : BOOL
VAR_INPUT
  pPoint : POINTER TO ST_DeformationPointAccurate;
END_VAR
VAR
  x_pos, dx_corr, dx_tmp : LREAL; // [m]
  y_pos, dy_corr, dy_tmp : LREAL; // [m]
END_VAR
// grid point position
x_pos := F_SubPixelToMeter(lPosSubPx:=FC_LREAL_TO_DINT(pPoint^.x_ref), fResSubPx:=_fPxResolution);  // [px -> m] 
y_pos := F_SubPixelToMeter(lPosSubPx:=FC_LREAL_TO_DINT(pPoint^.y_ref), fResSubPx:=_fPxResolution);  // [px -> m]
dx_corr := 0;
dy_corr := 0;

// calc - 4 point sheet deformation (PU and machine mechanical distortions)
IF _bEnable_4p THEN
  calc_4p_correction(x_pos:=x_pos, y_pos:=y_pos, dx_corr=>dx_tmp, dy_corr=>dy_tmp);
  dx_corr := dx_tmp + dx_corr;
  dy_corr := dy_tmp + dy_corr;
END_IF

IF _bEnablePuc_4p THEN  (*PUC 4P correction used*)
  calc_PUC_4p_correction(x_pos:=x_pos, y_pos:=y_pos, dx_corr=>dx_tmp, dy_corr=>dy_tmp);
  dx_corr := dx_tmp + dx_corr;
  dy_corr := dy_tmp + dy_corr;
END_IF

// calc - banana correction
IF _bEnable_banana THEN
  calc_banana_correction(x_pos:=x_pos, y_pos:=y_pos, fT1:=_fT1, fT2:=_fT2, dx_corr=>dx_tmp);
  dx_corr := dx_tmp + dx_corr;
END_IF
// apply new correction to deformation correction 
pPoint^.dx := pPoint^.dx + F_MeterToSubPixelReal(fPosMeter:=dx_corr, fResoSubPx:=_fPxResolution);
pPoint^.dy := pPoint^.dy + F_MeterToSubPixelReal(fPosMeter:=dy_corr, fResoSubPx:=_fPxResolution);

updateCorrection := TRUE;
END_METHOD

END_FUNCTION_BLOCK

// ---- POUs/Print/DefGrid/FB_PointCorr.TcPOU
FUNCTION_BLOCK FB_PointCorr
VAR PERSISTENT
  _fX_Pos, _fX_Ref : LREAL;   // x position (correction / reference)
  _fY_Pos, _fY_Ref : LREAL;   // y position (correction / reference)
END_VAR
VAR
  bCmd_X_minus : BOOL;    // command x minus
  bCmd_X_plus  : BOOL;    // command x plus
  bCmd_Y_minus : BOOL;    // command y minus
  bCmd_Y_plus  : BOOL;    // command y plus
  bAny         : BOOL;    // any pressed
  tSlow, tFast : TON;
  rTrig        : R_TRIG;
  nIncr        : LREAL;
  nBtnColor    : UDINT;
  // settings (init)
  _aName       : STRING(3);   // name of element
  _aUnit       : STRING(10);  // element intended [unit]
  _fX_Min, _fX_Max : LREAL;   // limit x
  _fY_Min, _fY_Max : LREAL;   // limit y
  _fIncrStep    : LREAL;      // incr. step slow (stay on button), fast *10
  _bButnInvertX, _bButnInvertY : BOOL;  // change buttons
  _bValInvertX, _bValInvertY   : BOOL;  // value *-1
END_VAR
VAR CONSTANT
  RED          : UDINT := 16#FFFF0000;
  GREEN        : UDINT := 16#FF00FF00;
END_VAR

bAny := bCmd_X_minus OR bCmd_X_plus OR bCmd_Y_minus OR bCmd_Y_plus;
rTrig(CLK:=bAny);
tSlow(IN:=bAny AND NOT tSlow.Q, PT:=T#500MS);
tFast(IN:=bAny AND NOT rTrig.Q, PT:=T#2S);

IF    tFast.Q AND tSlow.Q THEN nIncr := 10*_fIncrStep;
ELSIF tSlow.Q OR rTrig.Q THEN nIncr := _fIncrStep;
ELSE               nIncr := 0;
END_IF

nBtnColor := GREEN;
//    button pressed     increment +/-                show limit
IF    (bCmd_X_minus AND NOT _bButnInvertX) OR (bCmd_X_plus  AND _bButnInvertX) THEN _fX_Pos := _fX_Pos - nIncr; IF _fX_Pos<=_fX_Min THEN nBtnColor:=RED; END_IF
ELSIF (bCmd_X_plus  AND NOT _bButnInvertX) OR (bCmd_X_minus AND _bButnInvertX) THEN _fX_Pos := _fX_Pos + nIncr; IF _fX_Pos>=_fX_Max THEN nBtnColor:=RED; END_IF
ELSIF (bCmd_Y_minus AND NOT _bButnInvertY) OR (bCmd_Y_plus  AND _bButnInvertY) THEN _fY_Pos := _fY_Pos - nIncr; IF _fY_Pos<=_fY_Min THEN nBtnColor:=RED; END_IF
ELSIF (bCmd_Y_plus  AND NOT _bButnInvertY) OR (bCmd_Y_minus AND _bButnInvertY) THEN _fY_Pos := _fY_Pos + nIncr; IF _fY_Pos>=_fY_Max THEN nBtnColor:=RED; END_IF
END_IF

// apply limit
IF _fX_Pos<=_fX_Min THEN _fX_Pos:=_fX_Min; END_IF
IF _fX_Pos>=_fX_Max THEN _fX_Pos:=_fX_Max; END_IF
IF _fY_Pos<=_fY_Min THEN _fY_Pos:=_fY_Min; END_IF
IF _fY_Pos>=_fY_Max THEN _fY_Pos:=_fY_Max; END_IF

(*correction value in X*)
PROPERTY fX : LREAL
GET
fX := SEL(_bValInvertX, _fX_Pos, -1*_fX_Pos);
END_GET
SET
_fX_Pos := SEL(_bValInvertX, fX, -1*fX);
END_SET
END_PROPERTY

PROPERTY fX_Ref : LREAL
GET
fX_Ref := _fX_Ref;
END_GET
SET
_fX_Ref := fX_Ref;
END_SET
END_PROPERTY

(*correction value in Y*)
PROPERTY fY : LREAL
GET
fY := SEL(_bValInvertY, _fY_Pos, -1*_fY_Pos);
END_GET
SET
_fY_Pos := SEL(_bValInvertY, fY, -1*fY);
END_SET
END_PROPERTY

PROPERTY fY_Ref : LREAL
GET
fY_Ref := _fY_Ref;
END_GET
SET
_fY_Ref := fY_Ref;
END_SET
END_PROPERTY

METHOD init : BOOL
VAR_INPUT
  aName : STRING(3);       // name
  aUnit : STRING(10);      // display unit
  fX_Min, fX_Max : LREAL;  // Limits
  fY_Min, fY_Max : LREAL;  // Limits
  fIncrStep      : LREAL;  // Increment step (slow) VISU
  bButnInvertX, bButnInvertY : BOOL;  // change buttons
  bValInvertX,  bValInvertY  : BOOL;  // value *-1
END_VAR
_aName := aName;
_aUnit := aUnit;
_fX_Min := fX_Min; _fX_Max := fX_Max;
_fY_Min := fY_Min; _fY_Max := fY_Max;
_fIncrStep := fIncrStep;
_bButnInvertX := bButnInvertX;
_bButnInvertY := bButnInvertY;
_bValInvertX := bValInvertX;
_bValInvertY := bValInvertY;
END_METHOD

END_FUNCTION_BLOCK

// ---- POUs/Print/DefGrid/FB_PH_Grid.TcPOU
(*
  Specific printhead implementing the grid logic.
*)
FUNCTION_BLOCK FB_PH_Grid EXTENDS FB_PH IMPLEMENTS I_Correction_Grid
VAR
  // fifo queue
  fbFifo            : FB_GridPointFIFO;    // points fifo
  
  // queue status
  _bQueueBusy       : BOOL;               // point queue is not empty
  _bQueueError      : BOOL;               // point queue has an error

  // grid settings
  _bGridSet         : BOOL;               // grid is configured
  _nRows            : DINT;               // number of roi rows
  _nRowLowerBound, _nRowUpperBound : DINT;  //limites for roi rows of this ph
  _sDefGridSettings : ST_DefGridSettings;  // grid settings
  
  // checks
  _fbGetTaskIdx     : GETCURTASKINDEX;
  _taskIdx          : UDINT;
  _sTaskInfo        : PlcTaskSystemInfo;
  _lastCycle        : UDINT;
    
  // debug
  bEnSimPoints      : BOOL;               // enable grid point simulation
  bEnDebug          : BOOL;               // enable grid point history & point dump in logger
  nPointHead        : INT := 0;           // last list entry
  sPointHistory     : ARRAY[0..100] OF ST_GridPoint; // grid point history array
END_VAR

// sync points fifo to CB (PHs)
syncPoints();

// debug
IF bEnSimPoints THEN simPoints(); END_IF

PROPERTY bPointQueueBusy : BOOL
GET
bPointQueueBusy := SEL(fbFifo.nCount>0, FALSE, TRUE);   // busy as long queue is not empty
END_GET
END_PROPERTY

PROPERTY bPointQueueError : BOOL
GET
// check for errors
IF fbFifo.bError THEN
  _bQueueError := TRUE;
ELSE
  bPointQueueError := FALSE;
END_IF
END_GET
END_PROPERTY

(*
  Convert a point from DefGrid point to a GridPoint for hw write.
*)
METHOD PRIVATE convertPoint : ST_GridPoint
VAR_INPUT
  sPoint : POINTER TO ST_DeformationPoint;
  nPhPosY : DINT;
END_VAR
VAR
  nRoiOffset : DINT;
END_VAR
IF _sDefGridSettings.nGridPitchY = 0 THEN F_Report_Error(ErrType:=EN_REPORT_ERROR_TYPE.Report_Error_0Pointer); RETURN; END_IF

convertPoint.dx := DINT_TO_UINT(sPoint^.dx);
convertPoint.dy := DINT_TO_UINT(sPoint^.dy);

// variant1 with absolute Node address (based on number of grid-rows
(*convertPoint.node := 
  UDINT_TO_UINT(
      DINT_TO_UDINT(sPoint^.col)*sDefGridSettings.nGridSizeY 
    + DINT_TO_UDINT(sPoint^.row)
);*)

// variant2 - calculate FPGA ROI_address (roi_buffer address of grid point)
{warning 'TODO: update constants for calculation if FPGA is ok and make CONSTANTS'}
nRoiOffset := nPhPosY / TO_DINT(_sDefGridSettings.nGridPitchY);
convertPoint.node := TO_UINT((sPoint^.col MOD GVL_Deformation.nC_GridRoiCols) * GVL_Deformation.nC_GridRoiRows + sPoint^.row - nRoiOffset);
END_METHOD

(*
  Keep a history of last synced points.
*)
METHOD PRIVATE history
VAR_INPUT
  pPoint  : POINTER TO ST_GridPoint;
END_VAR
IF pPoint^.node = 0 THEN nPointHead := 0; END_IF  // internal reset on point address 0

sPointHistory[nPointHead] := pPoint^;
nPointHead := (nPointHead + 1) MOD 100;
END_METHOD

METHOD init : BOOL
VAR_INPUT
  aName                 : STRING;
  sPhDef                : ST_PH_DEF;                           (*ph definition structure*)
  tTempMonitor          : TIME;                                (*ph temperature monitoring timeout (warning after elapsed time)*)
  iFoeHandler           : I_FoeHandler;
  iChannel              : UDINT;  
  sCfgFolder            : T_MaxString;                          // path to config folder (where relative file name points to), keep='' if you have absolute paths in ads 

  bPositionX_Exist      : BOOL := TRUE; 
  aPositionX_Unit       : STRING := 'um'; 
  lPositionX_Min        : DINT := 0;  
  lPositionX_Max        : DINT := 1000;  
  bPositionY_Exist      : BOOL := TRUE;  
  aPositionY_Unit       : STRING := 'pixel';
  lPositionY_Min        : DINT := 0;  
  lPositionY_Max        : DINT := 100_000; 
  bShiftPositionX_Exist : BOOL := FALSE; 
  aShiftPositionX_Unit  : STRING := 'um'; 
  lShiftPositionX_Min   : DINT := 0;  
  lShiftPositionX_Max   : DINT := 1000;  
  bShiftPositionY_Exist : BOOL := FALSE;  
  aShiftPositionY_Unit  : STRING := 'pixel';
  lShiftPositionY_Min   : DINT := 0;  
  lShiftPositionY_Max   : DINT := 100_000; 
  bVoltageScale_Exist   : BOOL := TRUE;  
  aVoltageScale_Unit    : STRING := '%';
  fVoltageScale_Min     : REAL := 90.0;  
  fVoltageScale_Max     : REAL := 110.0; 
END_VAR
VAR
  bErr          : BOOL;
END_VAR
SUPER^.init(
  aName                 := aName,
  sPhDef                := sPhDef,
  tTempMonitor          := tTempMonitor,
  iFoeHandler           := iFoeHandler,
  iChannel              := iChannel,
  sCfgFolder            := sCfgFolder,
  bPositionX_Exist      := bPositionX_Exist,
  aPositionX_Unit       := aPositionX_Unit,
  lPositionX_Min        := lPositionX_Min,
  lPositionX_Max        := lPositionX_Max,
  bPositionY_Exist      := bPositionY_Exist,
  aPositionY_Unit       := aPositionY_Unit,
  lPositionY_Min        := lPositionY_Min,
  lPositionY_Max        := lPositionY_Max,
  bShiftPositionX_Exist := bShiftPositionX_Exist,
  aShiftPositionX_Unit  := aShiftPositionX_Unit,
  lShiftPositionX_Min   := lShiftPositionX_Min,
  lShiftPositionX_Max   := lShiftPositionX_Max,
  bShiftPositionY_Exist := bShiftPositionY_Exist,
  aShiftPositionY_Unit  := aShiftPositionY_Unit,
  lShiftPositionY_Min   := lShiftPositionY_Min,
  lShiftPositionY_Max   := lShiftPositionY_Max,
  bVoltageScale_Exist   := bVoltageScale_Exist,
  aVoltageScale_Unit    := aVoltageScale_Unit,
  fVoltageScale_Min     := fVoltageScale_Min,
  fVoltageScale_Max     := fVoltageScale_Max
);

nCorrection := 0;

_fbGetTaskIdx();
_taskIdx := _fbGetTaskIdx.index;
END_METHOD

(*
  Configure grid settings for ph.
*)
METHOD setGrid
VAR_INPUT
  sGrid : ST_DefGridSettings;
END_VAR
// grid settings checks
IF sGrid.nGridPitchX = 0 OR sGrid.nGridPitchY = 0 OR sGrid.nGridPoints = 0 THEN
  LogError('Invalid grid settings');
  RETURN;
END_IF

// store grid settings
_sDefGridSettings :=sGrid;

// caluclate roi row bounds
// lower row bound
_nRowLowerBound:=nPositionY / UDINT_TO_DINT(_sDefGridSettings.nGridPitchY);   // floor
_nRowLowerBound := LIMIT(0, _nRowLowerBound, UDINT_TO_DINT(_sDefGridSettings.nGridSizeY));  // limit to grid scope

// upper row bound
_nRowUpperBound:=(nPositionY + nHeadWidth) / UDINT_TO_DINT(_sDefGridSettings.nGridPitchY) + 1;
_nRowUpperBound := LIMIT(0, _nRowUpperBound, UDINT_TO_DINT(_sDefGridSettings.nGridSizeY));  // limit to grid scope

{warning 'TODO: update if RIO requirements are set by FPGA'}
// we just force to have 4 ROI rows and always charge effectively 4 row per head event if 3 would be sufficent
_nRowUpperBound := _nRowLowerBound + GVL_Deformation.nC_GridRoiRows - 1; 
// number of rows
_nRows := _nRowUpperBound - _nRowLowerBound + 1;

_bGridSet := TRUE;
END_METHOD

METHOD PRIVATE simPoints
VAR_INST
  tWrPoint      : TON := (PT:=T#1S);
  RandomNumber  : DRAND;
  sGridCfg    : ST_DefGridSettings := (nGridPitchX:=1024, nGridPitchY:=1024, nGridSizeX:=100, nGridSizeY:=100, nGridPoints:=10_000, nGridImageOffsetY:=0);   // some simulation defaults
  sNewPoint   : ST_DeformationPoint;
END_VAR
VAR
  random_val  : LREAL;
END_VAR
IF NOT _bGridSet THEN setGrid(sGrid:=sGridCfg); END_IF

// create and write a
tWrPoint(IN:=NOT tWrPoint.Q);
IF tWrPoint.Q THEN
  RandomNumber(Seed:=12, Num=>random_val);
  sNewPoint.dx := DINT_TO_UINT(FC_LREAL_TO_DINT((random_val * 100) - 50));
  RandomNumber(Seed:=12, Num=>random_val);
  sNewPoint.dy := DINT_TO_UINT(FC_LREAL_TO_DINT((random_val * 60) - 30));
  sNewPoint.col := sNewPoint.index / _nRows;
  sNewPoint.row := sNewPoint.index MOD _nRows + _nRowLowerBound;
  sNewPoint.index := (sNewPoint.index + 1) MOD 20;  // just 20 points
  writeCorrectionPoint(sPoint:=sNewPoint);
END_IF
END_METHOD

(*
  Sync deformation point to hardware.
*)
METHOD PRIVATE syncPoints
VAR
  sPoint  : ST_GridPoint;
  bOK     : BOOL;
  nPdiVal : ULINT;
END_VAR

IF fbFifo.nCount > 0 THEN
  bOK := fbFifo.Pop(sGridPoint=>sPoint);
  IF bOK THEN
    // build grid point pdi data
    nPdiVal     := UINT_TO_ULINT(sPoint.dx);
    nPdiVal     := nPdiVal OR SHL(UINT_TO_ULINT(sPoint.dy), 16);
    nPdiVal     := nPdiVal OR SHL(UINT_TO_ULINT(sPoint.node), 32);  
  
    sendCorrection(nCmdBit:=nC_CORRECTION_CMDBIT_GRIDPOINT, nData:=nPdiVal);

    //history
    IF bEnable AND bEnDebug THEN history(ADR(sPoint)); END_IF
  ELSE
    LogError('syncPoints: could not get a new GridPoint');
	END_IF
END_IF

// check for double calls within one task cycle
_sTaskInfo := TwinCAT_SystemInfoVarList._TaskInfo[_taskIdx];
IF _sTaskInfo.CycleCount = _lastCycle THEN
  LogError('syncPoints: was called twice in same task cycle');
END_IF
_lastCycle := _sTaskInfo.CycleCount;
END_METHOD

METHOD PRIVATE syncPoints_old
VAR
  sPoint  : ST_GridPoint;
  bOK     : BOOL;
  nPdiVal : ULINT;
END_VAR
nCorrection := nCorrection AND 16#0000FFFFFFFFFFFF;  // reset correction command only

IF fbFifo.nCount > 0 THEN
  bOK := fbFifo.Pop(sGridPoint=>sPoint);
  IF bOK THEN
    // build grid point pdi data
    nPdiVal     := UINT_TO_ULINT(sPoint.dx);
    nPdiVal     := nPdiVal OR SHL(UINT_TO_ULINT(sPoint.dy), 16);
    nPdiVal     := nPdiVal OR SHL(UINT_TO_ULINT(sPoint.node), 32);  
  
    // old sending (direct nCorrection access
    nCorrection := nCorrection AND 16#0000FFFFFFFFFFFF;  // reset correction command only
    nCorrection := SHL(1, 48) OR nPdiVal;      //set cmd [16bit] cmd / [48bit] of grid point in PDI var

    //history
    IF bEnable AND bEnDebug THEN history(ADR(sPoint)); END_IF
  ELSE
    LogError('syncPoints: could not get a new GridPoint');
	END_IF
END_IF
END_METHOD

(*
  Write a new Deformation Point to the hardware. 
  New added points will be synchroniced with the hardware with a FIFO queue.
  :return: TRUE on success
*)
METHOD writeCorrectionPoint : BOOL
VAR_INPUT
	(* add a new deformation point*)
	sPoint	: ST_DeformationPoint;
END_VAR
VAR
  sGridPoint : ST_GridPoint;
END_VAR
IF NOT _bGridSet THEN RETURN; END_IF

// filter points only for this head
IF sPoint.row >= _nRowLowerBound AND sPoint.row <= _nRowUpperBound THEN
  
  // convert deformation point to GridPoint for hw
  sGridPoint := convertPoint(sPoint:=ADR(sPoint), nPositionY);
  
  // add point
  writeCorrectionPoint := fbFifo.Push(sNewPoint:=sGridPoint);   // add new point

  IF bEnable AND bEnDebug THEN
    LogLvl(Lvl:=E_LogSeverity.Debug, Msg:=
      F_Concat4(
        'Write GridPoint '
        ,F_Concat4('c:', TO_STRING(sPoint.col), ' r:', TO_STRING(sPoint.row))
        ,F_Concat2(' -> node:', TO_STRING(sGridPoint.node))
        ,F_Concat4(' dx:', TO_STRING(sPoint.dx), ' dy:', TO_STRING(sPoint.dy))
      )
    );
  END_IF

END_IF
END_METHOD

END_FUNCTION_BLOCK

// ---- POUs/Print/DefGrid/FB_PH_Grid_Visu.TcPOU
FUNCTION_BLOCK FB_PH_Grid_Visu EXTENDS FB_VisuSelector
VAR_INPUT
END_VAR
VAR_OUTPUT
END_VAR
VAR_IN_OUT
  sI_Ary_Fb :   ARRAY[*] OF FB_PH_Grid;
END_VAR
VAR
  pL_Elem_Fb    : POINTER TO FB_PH_Grid;
END_VAR

(*checks*)
IF (ADR(sI_Ary_Fb) = 0) THEN
  F_Report_Error(Report_Error_0Pointer);
  RETURN;
END_IF

(*init fb*)
IF NOT bL_Init THEN
  SUPER^.setAryBounds(iLowerBoundary:=LOWER_BOUND(sI_Ary_Fb, 1), iUpperBoundary:=UPPER_BOUND(sI_Ary_Fb, 1));  
END_IF

(*call*)
SUPER^();
pL_Elem_Fb  := ADR(sI_Ary_Fb[pSelect^]);

END_FUNCTION_BLOCK

// ---- POUs/Print/DefGrid/FB_Pm_DMAX.TcPOU
(*
  Managing a production on a DigiRound machine.
*)
FUNCTION_BLOCK FB_Pm_DMAX EXTENDS FB_BasePrint IMPLEMENTS I_PrintStatusClient
VAR
 //references
  _pPU                : POINTER TO FB_PU;               (*PU reference*)
  _pAdsPU             : POINTER TO ST_ADS_PU;
  
  //settings
  _defaultPrintData   : ST_PRINT_SETTING;               (*default PDI data if no CT present*)
  _isVarData          : BOOL; 

  //status
  bPmActive           : BOOL;                           (*a production is active*)
  rfTrig_PmActive     : RF_TRIG;
  lastCreatedCT       : I_CT;                           (*last created container*)

  (*lists*)
  (*--list implementations*)
  prodList            : FB_ListPointerDyn;              (*list fb [pointer to I_CT] - current production elements*)
  _prodMem            : ARRAY[1..lNUM_LIST_SIZE] OF PVOID;   (*list memory for prodList*)
  (*--job trace list*)
  _currJobId          : STRING;                         (*id of current started job*)

  (*internals*)
  _pEcSrc : POINTER TO T_ErrSrc;                                    (*error source definition*)

END_VAR
VAR CONSTANT
  lNUM_LIST_SIZE        : DINT := iCPr_MAX_CONTAINER;   (*number of max. list elements*)
  // other logs
  aC_Dbg_NotReject      : STRING := 'could not rejectNext CT';
  aC_Dbg_InvPtrCT       : STRING := 'invalid pO_ContainerHead';
  aC_Dbg_InvPtrJob      : STRING := 'invalid Job pointer';
  aC_Ddb_GetNext        : STRING := 'getNext from: ';  
END_VAR

IF NOT bInitialized THEN RETURN; END_IF  // ignore

rfTrig_PmActive(CLK:=bPmActive);

(*
  Job was stopped. 
  :return: TRUE if some elements were aborted in machine.
*)
METHOD PRIVATE abortJob : BOOL
VAR
END_VAR
// a job stopped.

// NOTE: not implemented
END_METHOD

PROPERTY bReady : BOOL
GET
bReady := bPmActive;
END_GET
END_PROPERTY

PROPERTY bStarted : BOOL
GET
bStarted := rfTrig_PmActive.RT;
END_GET
END_PROPERTY

PROPERTY bStopped : BOOL
GET
bStopped := rfTrig_PmActive.FT;
END_GET
END_PROPERTY

(*
Create/Build a new container (CT) with next page to be printed.
*)
METHOD CT_Create : BOOL
VAR_INPUT
  sCT            : I_CT;                  // container to produce
END_VAR
VAR 
  _created       : BOOL := FALSE;
  sPage          : ST_PrintPageDef;
END_VAR
// prepare & checks
lastCreatedCT := 0;                      // invalidate last created
IF NOT bInitialized THEN RETURN; END_IF
IF sCT = 0 THEN LogError(aC_Dbg_InvPtrCT); RETURN; END_IF

(* getNext CT *)
IF getNext(sCT := sCT) THEN
  
  // define printer output
  sPage := sCT.sPageDef;
  IF    sPage.lType = EN_PrintPageType.maintenance THEN // - maintenance
    sCT.pCT^.lPrOutput := EN_PrinterOutput.trash;     // -> eject trash
  ELSIF sPage.lType = EN_PrintPageType.production OR   // - production
        sPage.lSrc = EN_PrintPageSrc.overprod OR       // - over-production
        sPage.lType = EN_PrintPageType.separator THEN  // - separator 
    sCT.pCT^.lPrOutput := EN_PrinterOutput.prod;      // -> production output
  ELSE                                                // - rest
    sCT.pCT^.lPrOutput := EN_PrinterOutput.trash;     // -> eject trash
  END_IF

  lastCreatedCT := sCT;                // successfully produced a CT, store last created CT (necessary for async access within this cycle)
  sCT.pCT^.bCreated := TRUE;
  _created := TRUE;
ELSE
  sCT.setError(EC_Print.ecPMInvGetNext, Src:=_pEcSrc^);   // getNext error
END_IF

(* logging *)
LogLvl(Lvl:=E_LogSeverity.Debug, Msg:=CONCAT('create CT: ', sCT.print(0)));

(*return value*)
CT_Create := _created;
END_METHOD

METHOD CT_Finish : BOOL
VAR_INPUT
  sCT            : I_CT;               // container to produce
  bSuccess       : BOOL;               // printed OK?
END_VAR
VAR
  bErr           : BOOL;
END_VAR
(* checks *)
IF NOT bInitialized THEN RETURN; END_IF                             // exit if no production is active
IF sCT = 0 THEN LogError(aC_Dbg_InvPtrCT); RETURN; END_IF  // log invalid pointer 

// remove from production list
IF NOT prodList.RemoveIndex(prodList.FindIndex(sCT.instance)) THEN
  LogError('CT_Finish: could not find CT in prodList'); 
END_IF

// tag machine errors on CT
IF sCT.pCT^.bValid AND NOT bSuccess THEN  
    sCT.setError(EC_Print.ecPMCTMachineErr, Src:=_pEcSrc^);            // tag CT with: error from machine 
END_IF

// report page done to PU
IF NOT sCT.pCT^.bReported AND sCT.pJob <> 0 THEN
  IF _pPU^.endPage(sCT:=sCT, bSuccess:=bSuccess) THEN
    ;
  ELSE
    sCT.setError(EC_Print.ecPMInvSet, Src:=_pEcSrc^);
  END_IF
END_IF

(* logging *)
IF bSuccess THEN
  LogLvl(Lvl:=E_LogSeverity.Detail, Msg:=CONCAT('successCT: ', sCT.print(0)));
ELSE
  LogLvl(Lvl:=E_LogSeverity.Detail, Msg:=CONCAT('eject  CT: ', sCT.print(0)));  
END_IF

(* return value *)
CT_Finish := TRUE;
END_METHOD

(*
  Finalize/Produce a CT. Now we shouldhave all necessary information for configuring the CT.
*)
METHOD CT_Produce : BOOL
VAR_INPUT
  sCT                 : I_CT;               // container to produce
END_VAR
VAR
  _produced           : BOOL := FALSE;
  sPage               : ST_PrintPageDef;
  bPresent            : BOOL;
END_VAR
(* parameter checks *)
IF NOT bInitialized THEN RETURN; END_IF
IF sCT = 0 THEN LogError(aC_Dbg_InvPtrCT); RETURN; END_IF

sCT.pCT^.bValid           := TRUE;                (* we have all data - CT is valid configured*)

// reject page if no container present or overproduction
sPage := sCT.sPageDef;
bPresent := sCT.pCT^.bProductPresent;
IF NOT bPresent AND sPage.lSrc <> EN_PrintPageSrc.overprod  THEN
  (*   add it to rejected queue (high prio reproduction), we will try to produce this CT in next cycle*)
  IF NOT _pPU^.rejPage(sCT:=sCT) THEN
    LogLvl(Lvl:=E_LogSeverity.Info, aC_Dbg_NotReject);
  END_IF
END_IF

(* logging *)
IF bPresent THEN LogLvl(Lvl:=E_LogSeverity.Detail,  Msg:=CONCAT('produceCT: ', sCT.print(0)));
            ELSE LogLvl(Lvl:=E_LogSeverity.Debug,   Msg:=CONCAT('produceCT: ', sCT.print(0))); END_IF

(* return value*)
CT_Produce := _produced;
END_METHOD

PROPERTY defaultPrData : ST_PRINT_SETTING
GET
defaultPrData := _defaultPrintData;
END_GET
END_PROPERTY

METHOD PRIVATE dynAddPage : BOOL
VAR_INPUT
  lType     : EN_PrintPageType; 
  lPageNr   : UDINT;
END_VAR
IF _pPU = 0 THEN F_Report_Error(ErrType:=EN_REPORT_ERROR_TYPE.Report_Error_0Pointer); RETURN; END_IF
IF lType <> EN_PrintPageType.maintenance THEN
  LogError('dynAddPage: only supports maintenance pages'); 
END_IF

_pPU^.addPage(lMaintPageNr:=lPageNr);
END_METHOD

(*
  get next page to be printed.
  :return:    TRUE if success.
*)
METHOD PRIVATE getNext : BOOL               (*get next image to be printed*)
VAR_INPUT
  sCT               : I_CT;                 (*container handle*)
END_VAR
VAR
  bErr              : BOOL;
  lRemainingPages   : UDINT;
END_VAR
VAR_INST
  rTrig_PreStop     : R_TRIG;
END_VAR
IF NOT bInitialized THEN RETURN; END_IF                    (* Exit if no production is active*)

// ask pu for a next page
bErr := NOT _pPU^.getPage(sCT:=sCT, lPagesLeft=>lRemainingPages);

// add to producing list
IF NOT prodList.AddItem(Item := sCT.instance) THEN 
  LogError('getNext: could not add CT to prodList');
  bErr := TRUE;
END_IF

getNext := NOT bErr;
END_METHOD

METHOD init : BOOL
VAR_INPUT
  pPU     : POINTER TO FB_PU;
  pAdsPU  : POINTER TO ST_ADS_PU;
  // machine specific
END_VAR
// parameter checks
IF pPU = 0 OR pAdsPU = 0 THEN
  F_Report_Error(ErrType:=EN_REPORT_ERROR_TYPE.Report_Error_0Pointer);
  RETURN;
END_IF

// register external references
_pPU := pPU;
_pAdsPU := pAdsPU;

// init lists
prodList(List:=_prodMem);  // initial call for list setup and init
prodList.Clear();

// init error source
_pEcSrc := ErrorCodes.fbErrCodeMngr.registerErrSource(
  nLocId:=0, 
  aInstPath:=InstanceName, 
  aLocDescr:='PrintManager DMAX'
);
IF _pEcSrc = 0 THEN LogError('could not register error source'); END_IF

//reset setates
bPmActive := FALSE;
lastCreatedCT := 0;

bInitialized := TRUE;
END_METHOD

METHOD JobFinished : BOOL
VAR_INPUT
  aSeparatorId   : STRING;
END_VAR
VAR
  pHandling      : POINTER TO ST_JobHandling;
END_VAR
// Job Handling -----------------------

// NOTE: nothing implemented for now
END_METHOD

PROPERTY lastCreated : I_CT
GET
lastCreated := lastCreatedCT;
END_GET
END_PROPERTY

METHOD mJobPause
END_METHOD

METHOD mJobStart
VAR_INPUT
	sJobDef	: I_JobDefinition;
END_VAR
VAR
  lCt     : UDINT;
  sHandling : ST_JobHandling;
  pHandling : POINTER TO ST_JobHandling;
END_VAR
IF NOT bInitialized THEN RETURN; END_IF
IF sJobDef = 0 THEN RETURN; END_IF

// start job 
LogLvl(lvl:=E_LogSeverity.Detail, Msg:=F_Concat5('PM start job: ', sJobDef.aJobId, ' (', sJobDef.aJobName, ')'));

// setup PrintManager with new job
_currJobId := sJobDef.aJobId;
_isVarData := sJobDef.isVarData();

// -- init last created
lastCreatedCT := 0;

// -- init defaultPrintData (TODO: not sure why we really need this)
MEMSET(ADR(_defaultPrintData), 0, SIZEOF(_defaultPrintData));   // reset default data

// -- add pre-production pages (product specific) -> maintenance pages
(*FOR lCt := 1 TO lStartEject DO 
  dynAddPage(lType:=EN_PrintPageType.maintenance, 1);
END_FOR*)

bPmActive := TRUE;
END_METHOD

METHOD mJobStop
VAR_INPUT
	sStatus	: I_JobStatus;
END_VAR
VAR
  eHandlingState  : EN_JobHandlingState;
END_VAR
IF NOT bInitialized THEN RETURN; END_IF

(*Stop job*)
LogLvl(lvl:=E_LogSeverity.Detail, Msg:=
  F_Concat7(
    'PM stop job P(',
    TO_STRING(sStatus.iJobProgress.lProductionCount), ') M(',
    TO_STRING(sStatus.iJobProgress.lMaintenanceCount), ') S(',
    TO_STRING(sStatus.iJobProgress.lScrapCount), ')'
  )
);

abortJob();

bPmActive := FALSE;
lastCreatedCT := 0;
END_METHOD

METHOD mProduced
VAR_INPUT
	(* current progress*)
	sProgress	: I_JobProgress;
END_VAR
IF NOT bInitialized THEN RETURN; END_IF
END_METHOD

END_FUNCTION_BLOCK

// ---- POUs/Print/DefGrid/FB_PrintOverview.TcPOU
FUNCTION_BLOCK FB_PrintOverview
VAR_INPUT
  fX_m,  fY_m   : LREAL;    // max. x/y position [m]
  nX_px, nY_px  : DINT;     // max. x/y pixel in view
  fPxToMRatio   : LREAL;    // 
  iPrintPosition : I_PrintPosition;
END_VAR

VAR
  // helper
  bInit   : BOOL;
  nCtr    : UDINT;
  nNum    : UDINT;
  
  // config
  _pCTM   : POINTER TO FB_CTManagerDefGrid;
  _pWorkerDefGrid : POINTER TO FB_WorkerDefGrid;
  _fPrintResolution : LREAL;      // [dpi]
  _fSubPixelResolution : LREAL;   // sub pixel resolution
  
  // Container view list
  iCT     : I_CT;
  aCTV    : ARRAY[1..iCPr_MAX_CONTAINER] OF FB_ContainerView;
  // Worker view list
  iWorker : I_Worker;
  aWorkerV: ARRAY[1..nC_MAX_WORKER_VIEWS] OF FB_ViewPositionControl;
  aWorkerFb: ARRAY[1..nC_MAX_WORKER_VIEWS] OF POINTER TO FB_WorkerDefGrid;
  
  // motion and position
  bMovingInd : BOOL;
  fSpeed  : LREAL;
  fbBlink : FB_BLINK;
  t : TIME;
  
  // last container debug
  nGridRowStart : UDINT;  // starting grid colum for Grid debug Visu
  nGridColStart : UDINT;  // starting grid colum for Grid debug Visu
  pLastCT : POINTER TO FB_ContainerDefGrid;   // pointer to last created container
  
  // time
  sCurrentDateTime : STRING;
  
  // view control
  bShowCtDetails : BOOL;
END_VAR
VAR CONSTANT
  nC_MAX_WORKER_VIEWS : UINT := 10;
END_VAR

IF NOT checkConfig() THEN RETURN; END_IF    // check config

// -- show CTs -----------------------
nNum := _pCTM^.nCount;
FOR nCtr := 1 TO nNum DO
  // get CT interface from list
  iCT := _pCTM^.getCT(nIdx:=nCtr);
  IF iCT <> 0 THEN
    // set position
    aCTV[nCtr].setPos(x:=iCT.GetPosRel(iTracker:=_pCTM^.iTracker), y:=0);

    // display
    aCTV[nCtr].bHide := FALSE;
    aCTV[nCtr]( iCT:=iCT, 
                iIdx:=UDINT_TO_UINT(iCT.pCT^.nMemIndex), 
                fPxtoMRatio:=fPxToMRatio, 
                fPosToMFactor := 0.0254 / (_fPrintResolution*_fSubPixelResolution), 
                iTracker:=_pCTM^.iTracker);
  END_IF
END_FOR

FOR nCtr := (nNum+1) TO iCPr_MAX_CONTAINER DO
  aCTV[nCtr].iCT := 0;
  aCTV[nCtr].bHide := TRUE;
END_FOR

// -- show Workers -----------------------
iWorker := _pWorkerDefGrid^.Root;
nCtr := 0;
WHILE iWorker <> 0 DO     // walk through worker chain
  nCtr := nCtr + 1;
  aWorkerFb[nCtr] := iWorker.Inst;  // get fb pointer
  aWorkerV[nCtr].bHide := FALSE;
  aWorkerV[nCtr].setPos(x:=aWorkerFb[nCtr]^.nTrackOffset, y:=0);
  iWorker:=iWorker.Next;
END_WHILE
FOR nCtr := (nCtr+1) TO nC_MAX_WORKER_VIEWS DO
  aWorkerV[nCtr].bHide := TRUE;
END_FOR

// -- show positioning -----------------------
fSpeed := iPrintPosition.getSpeed();
IF LrealIsNaN(x:=fSpeed) THEN
  fSpeed := 0;
END_IF
t := LREAL_TO_TIME(1000-fSpeed*900);
fbBlink(bI_Enable:=SEL(fSpeed > 0, FALSE, TRUE), tI_Time:=t, bO_Out=>bMovingInd);

// -- last container debug detail ------------
IF _pCTM^.nCount > 0 THEN
  iCT := _pCTM^.getCT(1);
  IF iCT <> 0 THEN  pLastCT := _pCTM^.GetContainerInstance(iCT:=iCT); END_IF
END_IF

// -- current time ---------------------------
sCurrentDateTime := F_TimeGetDateTime();

METHOD checkConfig : BOOL
VAR_INPUT
END_VAR
VAR_INST
  _fX_m, _fY_m   : LREAL;
  _nX_px, _nY_px : DINT; 
END_VAR
VAR
  bOK : BOOL;
END_VAR
IF NOT bInit THEN RETURN; END_IF
IF iPrintPosition = 0 THEN RETURN; END_IF

_fPrintResolution := iPrintPosition.fPrintResolution;
_fSubPixelResolution := iPrintPosition.fSubPxResolution;

// changed settings
IF _fX_m <> fX_m OR
          _fY_m <> fY_m OR
          _nX_px <> nX_px OR
          _nY_px <> nY_px THEN
  // save new config
   _fX_m := fX_m;
   _fY_m := fY_m;
   _nX_px := nX_px;
   _nY_px := nY_px;
   config();
END_IF

checkConfig := TRUE;
END_METHOD

METHOD PRIVATE config
VAR_INPUT
END_VAR
// NOTE: some config values are given only here (internally)
FOR nCtr := 1 TO iCPr_MAX_CONTAINER DO
  aCTV[nCtr].init(
    nXPosMin:=0,
    nXPosMax:= F_MeterToSubPixel(fPosMeter := fX_m, fResoSubPx := _fPrintResolution * _fSubPixelResolution),
    nYPosMin:=0,
    nYPosMax:=F_MeterToSubPixel(fPosMeter := fY_m, fResoSubPx := _fPrintResolution * _fSubPixelResolution),
    bXFlip:=TRUE,
    bYFlip:=FALSE,
    nXMinPx:=0,
    nXMaxPx:=nX_px,
    nYMinPx:=0,
    nYMaxPx:=nY_px,
  );
  aCTV[nCtr].setPos(x:=0, y:=0);
END_FOR
FOR nCtr := 1 TO nC_MAX_WORKER_VIEWS DO
  aWorkerV[nCtr].init(
    nXPosMin:=0,
    nXPosMax:= F_MeterToSubPixel(fPosMeter := fX_m, fResoSubPx := _fPrintResolution * _fSubPixelResolution),
    nYPosMin:=0,
    nYPosMax:=F_MeterToSubPixel(fPosMeter := fY_m, fResoSubPx := _fPrintResolution * _fSubPixelResolution),
    bXFlip:=TRUE,
    bYFlip:=FALSE,
    nXMinPx:=0,
    nXMaxPx:=nX_px,
    nYMinPx:=0,
    nYMaxPx:=nY_px,
  );
  aWorkerV[nCtr].setPos(x:=0, y:=0);
END_FOR

bInit := TRUE;
END_METHOD

METHOD init : BOOL
VAR_INPUT
  pCTM  : POINTER TO FB_CTManager;
  pWorkerDefGrid : POINTER TO FB_WorkerDefGrid;
END_VAR
IF pCTM = 0 OR pWorkerDefGrid = 0 THEN RETURN; END_IF

_pCTM := pCTM;
_pWorkerDefGrid := pWorkerDefGrid;

bInit := TRUE;
END_METHOD

END_FUNCTION_BLOCK

// ---- POUs/Print/DefGrid/FB_PrintPositionDmax.TcPOU
FUNCTION_BLOCK FB_PrintPositionDmax EXTENDS FB_BasePrint IMPLEMENTS I_Simulation
VAR_INPUT
  IlEncoderPulse      AT%I* : UDINT;                // Encoder counter intput
  IbEncoderWcState    AT%I* : BOOL;                 // Encoder EL5101 WcState
END_VAR
VAR_OUTPUT
  bStarted                  : BOOL;                 // position started moving
  bMoving                   : BOOL;                 // position is moving
END_VAR
// ----------------------------------
// configuration
VAR
  // configuration (init)
  _fPrintResolution         : LREAL := 600;         // print(head) resolution in [dpi]
  _fSubPxResolution         : LREAL := 32;          // SubPixel resolution [SubPx], resolution factor (fI_PrintResolution*fI_SubPxResolution=>Output resolution)
  _fTaskCycleTime           : LREAL := 0.002;        // Task cycle time in [s]
END_VAR
VAR PERSISTENT
  // config values changable during runtime (recipe, visu, property)
  _fEncoderResolution       : LREAL := 2.00475;     // Encoder resolution
  _bEnSpeedComp             : BOOL := FALSE;
  _fSpeedCompFactor         : LREAL := 0.0;         // TODO: define value
  _fSpeedCompRefSpeed       : LREAL := 0.0;         // TODO: define value
END_VAR
VAR CONSTANT
  fC_MinSpeed               : LREAL := 0.05;
END_VAR
// ---------------------------------
// internal variables
VAR
  // fb inst
  fbPositionMaster          : FB_PositionMaster;

  // internal vars
  fEncoderReso              : LREAL;                // used encoder resolution
  rTrigMoving               : R_TRIG;
  // simulation
  _bSim                     : BOOL;
  rfTrig_Sim                : RF_TRIG;
    
  // test functions
  (*bEnTestVsOld              : BOOL;    
  fbVencoder                : FB_V_ENCODER;
  Fb_Ph_Master              : FB_POSITION_MASTER;
  *)
END_VAR

rfTrig_Sim(CLK:=_bSim);
IF rfTrig_Sim.RT THEN SimEnter(); END_IF
IF rfTrig_Sim.FT THEN SimExit(); END_IF
IF _bSim THEN SimUpdate(); END_IF

// set internal used resolution
fEncoderReso := _fEncoderResolution;  

// compensate resolution (if enabled)
IF _bEnSpeedComp THEN
  fEncoderReso := F_EncoderSpeedComp(   
    fMasterSpeed:=fbPositionMaster.fMasterSpeed,
    fResolution:=fEncoderReso,
    fSpeedCompFactor:=_fSpeedCompFactor,
    fSpeedCompRefSpeed:=_fSpeedCompRefSpeed
  );
END_IF

// calc position / speed
fbPositionMaster(fResolutionInput:=fEncoderReso, lPosReference:=IlEncoderPulse);
// postion status
bMoving := fbPositionMaster.fMasterSpeed >= fC_MinSpeed; 
rTrigMoving(CLK:=bMoving);   // create started trigger output
bStarted := rTrigMoving.Q OR fbPositionMaster.bSyncReq;

PROPERTY bSimEnable : BOOL
GET
bSimEnable := _bSim;
END_GET
SET
_bSim := bSimEnable;
END_SET
END_PROPERTY

(*
  Get current "default" position.
  [SubPx] as return value and [um] as output
  :return: position in SubPx resolution
*)
METHOD getPosition : DINT
VAR_OUTPUT
  nPosition_px       : DINT;                 // Master position in [px]
  fPosition_um       : LREAL;                // Master position in [um]
END_VAR
getPosition := fbPositionMaster.lMasterPosition;
nPosition_px := fbPositionMaster.lMasterPosition / LREAL_TO_DINT(_fSubPxResolution);
fPosition_um := fbPositionMaster.fMasterPosition;
END_METHOD

(*
  Get "default" speed.
*)
METHOD getSpeed : LREAL
getSpeed := fbPositionMaster.fMasterSpeed;
END_METHOD

METHOD Init : BOOL
VAR_INPUT
  fPrintResolution    : LREAL := 600;         // print(head) resolution in [dpi]
  fSubPxResolution    : LREAL := 32;          // SubPixel resolution [SubPx], resolution factor (fI_PrintResolution*fI_SubPxResolution=>Output resolution)
  fTaskCycleTime      : LREAL;                 // Task cycle time in [s]
END_VAR
// store config
_fPrintResolution := fPrintResolution;
_fSubPxResolution := fSubPxResolution;
_fTaskCycleTime   := fTaskCycleTime;

// init fbs
// - position master
fbPositionMaster.init(
  fI_PrintResolution:=fPrintResolution, 
  fI_SubPxResolution:=fSubPxResolution, 
  fI_TaskCycleTime:=fTaskCycleTime, 
  bI_HWEncoder:=FALSE
);
END_METHOD

METHOD reset
VAR_INPUT
END_VAR
// reset positioning system
fbPositionMaster.reset();
END_METHOD

METHOD SimEnter : BOOL
_bSim := TRUE;
fbPositionMaster.bSim := TRUE;
END_METHOD

METHOD SimExit : BOOL
_bSim := FALSE;
fbPositionMaster.bSim := FALSE;
END_METHOD

METHOD SimUpdate : BOOL
//test_OldPhMaster(bEn:=bEnTestVsOld);
END_METHOD

END_FUNCTION_BLOCK

// ---- POUs/Print/DefGrid/F_EncoderSpeedComp.TcPOU
(*
  Encoder speed compensation.
  
  NOTE: Calculation can be disabled by setting fSpeedCompFactor=0
  :return: compensated encoder resolution
*)
FUNCTION F_EncoderSpeedComp : LREAL
VAR_INPUT
  (* live value *)
  fMasterSpeed                  : LREAL;		        (*Current Speed in [m/s]*)
  (* configuration *)
  fResolution                   : LREAL := 0.0;     (*default encoder resolution*)
  fSpeedCompFactor              : LREAL := 0.0;     (*TODO: define value*)
  fSpeedCompRefSpeed            : LREAL := 0.0;     (*TODO: define value*)
END_VAR
VAR
  fL_Compensation               : LREAL := 0.0;
END_VAR

IF (fSpeedCompFactor <> 0) AND (fMasterSpeed <> 0) THEN
  
  (*Calculate compensation*)
  fL_Compensation := (fMasterSpeed - fSpeedCompRefSpeed) * fSpeedCompFactor;
  fL_Compensation := DINT_TO_LREAL(FC_LREAL_TO_DINT(fL_Compensation * 10_000)) / 10_000;	(*Rounding to prevent small changes oscillation*)
  
  F_EncoderSpeedComp := fResolution * (1 + fL_Compensation);
ELSE
  
  (*return input resolution*)
  F_EncoderSpeedComp := fResolution;
END_IF;

END_FUNCTION

// ---- POUs/Print/DefGrid/FB_PS_Grid.TcPOU
FUNCTION_BLOCK FB_PS_Grid EXTENDS FB_PS_NewJetmap
VAR_INPUT
END_VAR
VAR_OUTPUT
END_VAR
VAR
  sCG : ARRAY[1..iCPr_NB_PH_PS_MAX] OF I_Correction_Grid;
  
  nRowMap : ARRAY[1..iCPr_NB_PH_PS_MAX,1..2] OF DINT; (*PH[x, [min, max]] Min..Max ROI row per head*)
  sDefGridSettings : ST_DefGridSettings;
END_VAR

METHOD newGridPoint : BOOL
VAR_INPUT
  sPoint : ST_DeformationPointAccurate;
END_VAR
VAR
  bOK : BOOL;
  bLimited : BOOL;
  i : UDINT;
  sPointPx : ST_DeformationPoint;
END_VAR
// write to head(s)
FOR i:=1 TO nPh DO
  
  //Check if point in scope of printhead (rows) (NOTE: could be remo)
  IF sPoint.row >= nRowMap[i,1] AND sPoint.row <= nRowMap[i,2] THEN

    // write DefGrid point
    sPointPx := F_EncodeDeformationPoint(sPoint:=sPoint, nResolution:=1);   // convert point to fixed point (floor)
    bOK := sCG[i].writeCorrectionPoint(sPoint:=sPointPx);
    IF NOT bOK THEN 
      LogWarning(F_Concat6('Could not write GridPoint to PH[', TO_STRING(i), '] c:', TO_STRING(sPoint.col), '/r:', TO_STRING(sPoint.row)));
    END_IF
	END_IF
END_FOR

newGridPoint := TRUE;
END_METHOD

METHOD printPrepare
VAR_OUTPUT
  bNoHeadEnabled : BOOL;
  bPrepareError  : BOOL;
END_VAR
VAR
  i : UDINT;
  bEn : BOOL;
END_VAR
SUPER^.printPrepare(bNoHeadEnabled=>bNoHeadEnabled, bPrepareError=>bPrepareError);
END_METHOD

METHOD registerCG : BOOL
VAR_INPUT
      iNewPh : I_PH;                // printhead interface
      iNewCG : I_Correction_Grid;   // correction grid interface
END_VAR
IF iNewCG = 0 OR iNewCG = 0 THEN LogError('registerCG: Invalid parameter'); F_Report_Error(ErrType:=EN_REPORT_ERROR_TYPE.Report_Error_0Pointer); RETURN; END_IF
IF THIS^.registerPh(iNewPh:=iNewPh) THEN
    sCG[nPh] := iNewCG; //add CG same as printhead, they are in sync
END_IF
END_METHOD

METHOD setGrid
VAR_INPUT
  sGrid : ST_DefGridSettings;
END_VAR
VAR
  i : UDINT;
END_VAR
// grid settings checks
IF sGrid.nGridPitchX = 0 OR sGrid.nGridPitchY = 0 OR sGrid.nGridPoints = 0 THEN
  LogError('Invalid grid settings');
  RETURN;
END_IF

// save grid settings
sDefGridSettings :=sGrid;

// set grid on PH 
FOR i:=1 TO nPh DO
  sCG[i].setGrid(sGrid:=sGrid);
  
  (* setup grid filter in PS (for better performance, pre-filter points before sending to ph) 
      this could removed so we have the RIO calculation only once.*)
  IF sPh[i] <> 0 AND sCG[i] <> 0 THEN
    // lower row bound
    nRowMap[i,1]:=sPh[i].nPositionY / UDINT_TO_DINT(sDefGridSettings.nGridPitchY);   // floor
    // upper row bound
    nRowMap[i,2]:=(sPh[i].nPositionY + sPh[i].nHeadWidth) / UDINT_TO_DINT(sDefGridSettings.nGridPitchY) + 1;
    {warning 'TODO: review with RIO calculation if FPGA is right'}
    nRowMap[i,2]:=nRowMap[i,1] + GVL_Deformation.nC_GridRoiRows - 1;
    
    // limit to grid scope
    nRowMap[i,1] := LIMIT(0,nRowMap[i,1],UDINT_TO_DINT(sDefGridSettings.nGridSizeY));
    nRowMap[i,2] := LIMIT(0,nRowMap[i,2],UDINT_TO_DINT(sDefGridSettings.nGridSizeY));
  ELSE
    F_Report_Error(ErrType:=EN_REPORT_ERROR_TYPE.Report_Error_0Pointer);
  END_IF  
END_FOR
END_METHOD

END_FUNCTION_BLOCK

// ---- POUs/Print/DefGrid/FB_PythonInterface.TcPOU
FUNCTION_BLOCK FB_PythonInterface EXTENDS T_NamedBase
VAR
  // interface paths (config)
  sPythonInterfacePath : STRING(255); //e.g. 'PRG_x.fb_PythonInterface'
  sPythonContainerPath : STRING(255); //e.g. 'PRG_x.fb_ContainerManager.sL_Containers[%id%].fb_ImageDeformation'
  sPythonScriptPath    : STRING(255);

	bPythonHeartbeat : BOOL;      // <- script is toggling this value as long as it's alive (for plc watchdog of script)
	nPythonPID : UDINT := 0;      // <- python process id (evaluated and given by external script)
  nPythonNewJob : DINT;         // -> new job indication to script
  bPythonNewJobDone : BOOL;     // <- new job registered/done by script

	nContainerToRegister : DINT := -1; // <- triggers a new container creation, except if < 0
  nContainerToRegister_mem : DINT := -1;
	nContainerToDelete : DINT := -1;   // <- triggers a new container deletion, except if < 0
  nContainerToDelete_mem : DINT := -1;
  
  // job definition
  aPythonJobName : T_MaxString; // -> new job name
  aPythonJobGuid : T_MaxString; // -> new job GUID
  //Job settings all in [px]
  nPythonImageOffsetY : UDINT := 0;     // [px]  y offset from 0 to source image
  nPythonImageWidth : UDINT := 1000;    // [px]  source image width (depth)
  nPythonImageHeight  : UDINT := 1000;  // [px]  source image height (width)
  //Grid settings
  nPythonGridPitchX  : UDINT := 100;    // [px]
  nPythonGridPitchY  : UDINT := 100;    // [px]
  nPythonGridSizeX   : UDINT := 0;      // (not yet used) number of grid columns
  nPythonGridSizeY   : UDINT := 0;      // (not yet used) number of grid rows
  //Cam specific settings
  nPythonCamFrameWidth  : UDINT := 200; // [px]
  
  nState : UDINT;
  fbStateTimer : TON;
  fBScriptLauncher : FB_ScriptLauncher;
  _bEnable : BOOL;
  _bKeepAlive : BOOL := TRUE; // keep script alive (restart after crash/close)
  _nStarts : UDINT;   // number of script start attempts
  _nErrCtr : UDINT;   // script error state counter
  _bBusy : BOOL;
  _nErrId : UDINT;
  _bJobStartRequest: BOOL;
  _bJobStopRequest: BOOL;
  _bResetError : BOOL;    // reset state machine error 
  _nJobIdCtr : DINT;
 
	// Python script heartbeat
	fbWatchdog : TOF;
	tWatchdogPeriod : TIME := T#1S;
	fbHeartbeat1 : R_TRIG;
	fbHeartbeat2 : F_TRIG;
	bScriptAlive : BOOL;

END_VAR

VAR CONSTANT
  cStateIdle      : UDINT := 0;
  cStateStartup   : UDINT := 10;
  cStartScript    : UDINT := 20;
  cStateRunning   : UDINT := 30;
  cStateJobActive : UDINT := 40;
  cStateError     : UDINT := 50;
  cStateStop      : UDINT := 60;
  cStateStopping  : UDINT := 70;
  
  cMaxStartAttempts : UDINT := 5;
END_VAR

InterfaceStateMachine();

// reset Container commands, so we suer have a change event on index
IF nContainerToRegister >= 0 AND nContainerToRegister_mem >= 0 THEN nContainerToRegister := -1; END_IF
IF nContainerToDelete >= 0 AND nContainerToDelete_mem >= 0 THEN nContainerToDelete := -1; END_IF
nContainerToRegister_mem := nContainerToRegister;
nContainerToDelete_mem := nContainerToDelete;

fbHeartbeat1(CLK := bPythonHeartbeat);
fbHeartbeat2(CLK := bPythonHeartbeat);
fbWatchdog(IN := fbHeartbeat1.Q OR fbHeartbeat2.Q, PT:=tWatchdogPeriod);
bScriptAlive := fbWatchdog.Q AND nPythonPID <> 0;

METHOD ackError
VAR_INPUT
END_VAR
_bResetError := TRUE;
END_METHOD

{attribute 'monitoring':='call'}
PROPERTY bBusy : BOOL
GET
bBusy := _bBusy;
END_GET
END_PROPERTY

PROPERTY bEnable : BOOL
GET
bEnable := _bEnable;
END_GET
SET
_bEnable := bEnable;
END_SET
END_PROPERTY

{attribute 'monitoring':='call'}
PROPERTY bError : BOOL
GET
IF nState = cStateError THEN bError := TRUE; END_IF;
END_GET
END_PROPERTY

{attribute 'monitoring':='call'}
PROPERTY bJobActive : BOOL
GET
IF nState = cStateJobActive THEN bJobActive := TRUE; END_IF;
END_GET
END_PROPERTY

{attribute 'monitoring':='call'}
PROPERTY bRunning : BOOL
GET
IF nState = cStateRunning THEN bRunning := TRUE; END_IF;
END_GET
END_PROPERTY

METHOD Init : BOOL
VAR_INPUT
  sCTManagerPath : T_MaxString;  // ct manager path (plc variable instance path)
  sScriptPath    : T_MaxString;  // path to python script base folder, e.g. C:\Work\script
END_VAR
sPythonInterfacePath := THIS^.InstanceName;
sPythonContainerPath := sCTManagerPath;
sPythonScriptPath    := sScriptPath;

// init launcher
fBScriptLauncher.Init(sPythonScriptPath);

// some variable init
aPythonJobName := 'JobNameUnknown';
aPythonJobGuid := 'aaaaaaaa-bbbb-cccc-dddd-eeeeeeeeeeee';

//Launch init procedure
fbStateTimer(PT:=T#5S);
nState := cStateIdle;
END_METHOD

ACTION InterfaceStateMachine:

CASE(nState) OF
  // Idle
  cStateIdle  :
    _bJobStartRequest:=FALSE;
    _bJobStopRequest:=FALSE;
    _bResetError := FALSE;
    IF bEnable THEN
      nState := cStateStartup;
    END_IF  

  //Startup
  cStateStartup   :
    fbStateTimer(IN:=TRUE);         // start timeout
    _bBusy := TRUE;

    IF fbStateTimer.Q THEN
      fbStateTimer(IN:=FALSE);
      _nStarts := _nStarts + 1;
      IF bScriptAlive THEN
        nState := cStateRunning;    // is already running
      ELSE  
        RunPythonScript();          // start script
        nState := cStartScript;
			END_IF
		END_IF
  
  //Start Python script and wait until it starts
  cStartScript    :
    fbStateTimer(IN:=TRUE);
    _bBusy := TRUE;

    IF NOT fBScriptLauncher.bBusy AND bScriptAlive THEN 
      IF fBScriptLauncher.bError THEN //Launch error
        LogError(F_Concat2('Script start error=', TO_STRING(fBScriptLauncher.nErrId)));
        nState := cStateError;
      ELSE //Launch done and heartbeat ok
        nState := cStateRunning;
        fbStateTimer(IN:=FALSE);
			END_IF
    ELSIF fbStateTimer.Q THEN //Timeout error (could not start)
      IF fBScriptLauncher.bError THEN //Launch error
        ///LogError(F_Concat2('Script start error=', TO_STRING(fBScriptLauncher.nErrId)));
        LogError(F_Concat2('Script start error=', F_GetAdsErrStr(fBScriptLauncher.nErrId)));
      ELSE
        LogError('Script start error');
      END_IF
      nState := cStateError;
		END_IF
 
  //Script running with correct watchdog feedback
  cStateRunning   : 
    fbStateTimer(IN:=_bJobStartRequest);
    _bBusy := _bJobStartRequest;
    _bJobStopRequest := FALSE;
    _nStarts := 0;
    
    IF _bJobStartRequest AND bPythonNewJobDone THEN
      _bJobStartRequest:=FALSE;
      bPythonNewJobDone := FALSE; 
      fbStateTimer(IN:=FALSE);  
      nState := cStateJobActive;
    ELSIF NOT bScriptAlive THEN //Watchdog error
      LogError('Script watchdog error');
      nState := cStateError;
    ELSIF fbStateTimer.Q THEN //Job timeout error
      LogError('Script new job done error');
      nState := cStateError;
    ELSIF NOT bEnable THEN
      nState := cStateStop;
		END_IF
  
  //JobStarted
  cStateJobActive :
    fbStateTimer(IN:=_bJobStopRequest);
    _bBusy := _bJobStopRequest;
    
    IF _bJobStopRequest THEN
      nPythonNewJob := 0;
    END_IF;  
    
    IF _bJobStopRequest THEN
      _bJobStopRequest:=FALSE;
      fbStateTimer(IN:=FALSE);  
      nState := cStateRunning;
    ELSIF NOT bScriptAlive THEN //Watchdog error
      LogError('Script watchdog error');
      nState := cStateError;
    ELSIF fbStateTimer.Q THEN //Job timeout error
      LogError('Script new job done error');
      nState := cStateError;
    ELSIF NOT bEnable THEN
      nState := cStateStop;
		END_IF
  
  //Error  
  cStateError     :
    fbStateTimer(IN:=FALSE);  
    _bJobStartRequest:=FALSE;
    _bJobStopRequest:=FALSE;
    // reset error 
    IF _bResetError THEN
      _nStarts := 0;          // exit error 
      _nErrCtr := _nErrCtr + 1;
      nState := cStateStop ;
    ELSIF NOT bEnable THEN
      nState := cStateStop ;  // just stop
    ELSIF (_bKeepAlive AND _nStarts <= cMaxStartAttempts)  THEN
      _nErrCtr := _nErrCtr + 1;   // retry 
      nState := cStateStop ;
		END_IF
    
  //Stop 
  cStateStop  :
    StopPythonScript();
    nState := cStateStopping;

  // Stopping
  cStateStopping  :
    IF NOT fBScriptLauncher.bBusy THEN 
      IF fBScriptLauncher.bError THEN //Launch error
        LogError(F_Concat2('Script stop errror:', TO_STRING(fBScriptLauncher.nErrId)));
			END_IF
      nState := cStateIdle;
    END_IF

END_CASE
END_ACTION

METHOD JobStart
VAR_INPUT
  aJobName       : T_MaxString;
  aJobGuid       : T_MaxString;
  nJobImageWidth : UDINT;
  nJobImageHeigth  : UDINT;
  nCamFrameWidth : UDINT;
  pGridSettings  : POINTER TO ST_DefGridSettings;
END_VAR
_bJobStartRequest := TRUE;
_nJobIdCtr := _nJobIdCtr + 1;
nPythonNewJob := _nJobIdCtr;

aPythonJobName := aJobName;
aPythonJobGuid := aJobGuid;
nPythonImageWidth := nJobImageWidth * GVL_Deformation.nC_GridSubReso;
nPythonImageHeight :=nJobImageHeigth * GVL_Deformation.nC_GridSubReso;
nPythonCamFrameWidth := nCamFrameWidth * GVL_Deformation.nC_GridSubReso;
IF pGridSettings <> 0 THEN
  nPythonImageOffsetY := pGridSettings^.nGridImageOffsetY * GVL_Deformation.nC_GridSubReso;
  nPythonGridPitchX := pGridSettings^.nGridPitchX * GVL_Deformation.nC_GridSubReso;
  nPythonGridPitchY := pGridSettings^.nGridPitchY * GVL_Deformation.nC_GridSubReso;
  nPythonGridSizeX := pGridSettings^.nGridSizeX * GVL_Deformation.nC_GridSubReso;
  nPythonGridSizeY := pGridSettings^.nGridSizeY * GVL_Deformation.nC_GridSubReso; 
END_IF
END_METHOD

METHOD JobStop : BOOL
VAR_INPUT
END_VAR
_bJobStopRequest:=TRUE;
END_METHOD

{attribute 'monitoring':='call'}
PROPERTY nErrorId : UDINT
GET
nErrorId := _nErrId;
END_GET
END_PROPERTY

(*
  Register CT to script.
  :return: TRUE if success.
*)
METHOD RegisterCT : BOOL
VAR_INPUT
  nCTIdx  : UDINT;  // ct memory index
END_VAR
IF NOT bScriptAlive THEN RETURN; END_IF  // script not ready, ignore request

nContainerToRegister := UDINT_TO_DINT(nCTIdx);
RegisterCT := TRUE;
END_METHOD

METHOD RemoveCT : BOOL
VAR_INPUT
    nCTID : UDINT;
END_VAR
IF NOT bScriptAlive THEN RETURN; END_IF  // script not ready, ignore request

nContainerToDelete := UDINT_TO_DINT(nCTID);

RemoveCT := TRUE;
END_METHOD

METHOD PRIVATE RunPythonScript : BOOL
VAR_INPUT
END_VAR
VAR
  ams_host : STRING;
  ams_port : UINT;
  cmd : STRING;
END_VAR
// config launcher cmd line for script
//   e.g. fBScriptLauncher.Start('172.17.7.143.1.1 851 PRG_PRINT.fbWorkerDefGrid_Python.fbPythonInterface --sim_mode');

// get parameter dynamically
ams_host := PRG_SYSTEMBASE.sO_AmsNetIdLocalHost;  // localhost
ams_port := TwinCAT_SystemInfoVarList._AppInfo.AdsPort;
cmd := F_Concat5(ams_host,' ',TO_STRING(ams_port),' ',sPythonInterfacePath);
fBScriptLauncher.sStartScriptName := 'start.bat';
fBScriptLauncher.sStopScriptName  := 'stop.bat';
fBScriptLauncher.Start(cmd);
END_METHOD

METHOD PRIVATE StopPythonScript
VAR_INPUT
END_VAR
fBScriptLauncher.Stop(nPID := THIS^.nPythonPID);
END_METHOD

{attribute 'monitoring':='call'}
PROPERTY tWatchdogTime : TIME
GET
tWatchdogTime := fbWatchdog.ET;
END_GET
END_PROPERTY

END_FUNCTION_BLOCK

// ---- POUs/Print/DefGrid/FB_StartPositionDummy.TcPOU
(*
  A start position detection function block dummy.
  A dummy implementation to simulate start triggers at desired positions.
*)
FUNCTION_BLOCK FB_StartPositionDummy EXTENDS FB_BasePrint IMPLEMENTS I_StartPosDetect, I_PrintStatusClient, I_Sim
VAR_INPUT
  bTrigger                    : BOOL;       // manual trigger
  lPosition                   : DINT;       // current position [SubPx]
  fSpeed                      : LREAL;      // current speed [m/s]
  fResolution                 : LREAL;      // current print resolution [dpi*SubPx]
END_VAR

VAR
  // properties
  _bSim               : BOOL;       // simulatio mode active (PROPERTY)
  _bCreateTrigger     : BOOL;       // create new CT trigger (PROPERTY)
  _nStartPosX0        : DINT;       // create position for CT (absolut) [SubPx] (PROPERTY)
  _bAutoTrigger       : BOOL;       // automatic sheet triggers
  
  // config
  iJobDefinition      : CalmarCompPrint.I_JobDefinition;
  
  // local helper
  rfNewCT             : RF_TRIG;    // trigger new ct
  nSheetLength        : DINT;       // sheet length in [SubPx]
  nSheetGap           : DINT;       // sheet gap in [SubPx]
  nSheetEndPosition   : DINT;       // sheet end position [SubPx]
  nNextSheetPosition  : DINT;       // next trigger location
  fSheetPerHour       : LREAL;      // sheets per hour
  fSheetSpeed         : LREAL;      // [m/min] speed meter per minute
  tCheckTrigger       : TON;
  
  tCurrentTimeStamp   : T_DCTIME64; // get current timestamp
  fCurrentTimeStamp   : LREAL;      // current timestamp
  fSensorTimeStamp    : LREAL;      // sensor timestamp
  fDeltaDistance      : LREAL;      // distance that the substrate moved between the detection and the treatment of the information [m]
  
  rfTrig_Sim          : RF_TRIG;
END_VAR

VAR PERSISTENT
  // simulation configuration
  fSheetLength   : LREAL := 0.5;    // [m] sheet length (local or per job given)
  fSheetGap      : LREAL := 0.12;   // [m] gap between two sheets
END_VAR

// checks and fixes
IF iJobDefinition = 0 THEN RETURN; END_IF
IF fSpeed = 0 THEN RETURN; END_IF
IF fSheetLength = 0 THEN fSheetLength := 1; END_IF
IF fResolution = 0 THEN fResolution := 600*32; END_IF
rfTrig_Sim(CLK:=_bSim);
IF    rfTrig_Sim.RT THEN SimEnter(); 
ELSIF rfTrig_Sim.FT THEN SimExit(); END_IF

IF NOT _bSim THEN RETURN; END_IF

// calculations
fSheetSpeed := fSpeed * 60;  // [m/s] -> [m/min]
nSheetGap := F_MeterToSubPixel(fPosMeter := fSheetGap, fResoSubPx := fResolution);  // [m] -> [SubPx]
fSheetPerHour := (60*60)/((fSheetLength+fSheetGap)/fSpeed);
nSheetLength := F_MeterToSubPixel(fPosMeter := fSheetLength, fResoSubPx := fResolution);  // [mm] -> [SubPx]
nNextSheetPosition := _nStartPosX0 + nSheetLength + nSheetGap; 
tCheckTrigger(PT:=TO_TIME(((fSheetLength+fSheetGap)/fSpeed)*1000));

// internal trigger creation
IF (lPosition - nNextSheetPosition) > 0 AND _bAutoTrigger THEN
  bTrigger := TRUE;
  tCheckTrigger(IN:=FALSE);
  tCheckTrigger(IN:=TRUE);
END_IF

// on trigger
rfNewCT(CLK := bTrigger, RT => _bCreateTrigger);
IF _bCreateTrigger THEN   // new ct created
  bTrigger := FALSE;  // reset trigger
  
  (* Calculate the current and sensor time stamp (keep old code not really necessary because we use current timestamp)*)
  tCurrentTimeStamp := F_GetCurDcTaskTime64();
  fCurrentTimeStamp := (ULINT_TO_LREAL(tCurrentTimeStamp )) / 1_000_000.0; (*in ms*)
  fSensorTimeStamp  := fCurrentTimeStamp;
  fDeltaDistance := (fCurrentTimeStamp - fSensorTimeStamp) * 0.001 * fSpeed;  (*Distance that the substrate moved between the detection and the treatment of the information [m]*)
  
  // sheet start and sheet end pos in [SubPx]
  _nStartPosX0     := lPosition - F_MeterToSubPixel(fPosMeter := fDeltaDistance, fResoSubPx := fResolution);
  nSheetEndPosition := _nStartPosX0 + nSheetLength;
END_IF

{attribute 'monitoring' := 'call'}
(*Simulation is enabled set/get*)
PROPERTY bSimEnable : BOOL
GET
bSimEnable := _bSim;
END_GET
SET
_bSim := bSimEnable;
END_SET
END_PROPERTY

(*
  A new container detected.
  NOTE: a pulse only
*)
PROPERTY bStartTrig : BOOL
GET
bStartTrig := _bCreateTrigger;
END_GET
END_PROPERTY

(*
  A valid container detected.
*)
PROPERTY bValid : BOOL
GET
bValid := TRUE;
END_GET
END_PROPERTY

METHOD mJobPause
END_METHOD

METHOD mJobStart
VAR_INPUT
	sJobDef	: CalmarCompPrint.I_JobDefinition;
END_VAR
IF sJobDef = 0 THEN LogError('JobStart: no sJobDef given'); RETURN; END_IF

iJobDefinition := sJobDef;    // current job definition
fSheetLength := iJobDefinition.fSubstrateDepth;
END_METHOD

